// TwinCAT 3 PLC project mover_demo
// ProgramVersion: 3.1.4024.12
// libraries:
//   CmpBitmapPool, * (System)
//   Tc2_Math, * (Beckhoff Automation GmbH)
//   Tc2_MC2, * (Beckhoff Automation GmbH)
//   Tc2_MC2_Drive, * (Beckhoff Automation GmbH)
//   Tc2_Standard, * (Beckhoff Automation GmbH)
//   Tc2_System, * (Beckhoff Automation GmbH)
//   Tc2_Utilities, * (Beckhoff Automation GmbH)
//   Tc3_JsonXml, * (Beckhoff Automation GmbH)
//   Tc3_Module, * (Beckhoff Automation GmbH)
//   VisuDialogs, * (System)
//   VisuSymbols,3.5.10.0,System
// project tree:
//   DUTs/Helptec/Axis/ AxisBase_t.TcDUT (not stored), AxisBeckhoff_t.TcDUT (not stored), AxisLinMotConst_t.TcDUT, AxisLinMot_t.TcDUT (not stored), AxisSMC_t.TcDUT, typeInputArea.TcDUT, typeOutputArea.TcDUT (not stored)
//   DUTs/Helptec/ Cylinder2Pos_config.TcDUT (not stored), enLamp.TcDUT (not stored), enState.TcDUT (not stored), structAlarm.TcDUT (not stored), structButton.TcDUT (not stored)
//   DUTs/Helptec/Recipe/ RecipeAxisLinear2Pos_t.TcDUT (not stored)
//   DUTs/Helptec/RS_Axis/ FeederDelays_t.TcDUT, MoveProfile1D_t.TcDUT, MoveProfile_t.TcDUT (not stored), TriggerType_e.TcDUT (not stored), VectorMove1D_t.TcDUT (not stored)
//   DUTs/ PieceType_e.TcTLEO (not stored), Mover_st.TcDUT (not stored), Piece_st.TcDUT (not stored)
//   / GlobalTextList.TcGTLO (not stored) (excluded from build), PlcTask.TcTTO, Visualization Manager.TcVMO (not stored), VISU_TASK.TcTTO (not stored)
//   GVLs/ AXIS.TcGVL, CONST.TcGVL (not stored), GVL.TcGVL (not stored), HMI.TcGVL, IN.TcGVL (not stored), IO_BOX.TcGVL, OUT.TcGVL (not stored), PERS.TcGVL (not stored), SIMU.TcGVL (not stored)
//   POUs/00_MAIN/ DEBUG.TcPOU, MAIN.TcPOU, _02_SAFETY.TcPOU, _05_FLAGS.TcPOU (not stored)
//   POUs/00_MAIN/FB%27s/ FB_Safety.TcPOU (not stored)
//   POUs/10_HMI/FB%27s/ FB_BUTTON.TcPOU (not stored), FB_HMI_BT.TcPOU (not stored), FB_Keba_key.TcPOU (not stored), FB_LampeBNI007F.TcPOU (not stored), FB_STATE.TcPOU (not stored)
//   POUs/10_HMI/ _10_HMI.TcPOU (not stored), _11_PAR_CHK.TcPOU (not stored), _14_STATE.TcPOU (not stored)
//   POUs/20_AUTO/ Axis_e.TcTLEO, LinearAxis_e.TcTLEO (not stored), RecipeType_e.TcTLEO, Recipe_21_101_t.TcDUT (not stored), StationList_e.TcTLEO (not stored), _20_AUTO.TcPOU (not stored), _21_CopyDefaultRecipe.TcPOU (not stored)
//   POUs/20_AUTO/BuR SuperTrack com/ CT_Shuttle_BR_to_Tc_Status_t.TcDUT (not stored), CT_Shuttle_BR_to_Tc_t.TcDUT (not stored), CT_Shuttle_BR_to_Tc_u.TcDUT (not stored), CT_Shuttle_Tc_To_BR_Command_t.TcDUT (not stored), CT_Shuttle_Tc_to_BR_t.TcDUT, CT_Shuttle_Tc_to_BR_u.TcDUT, CT_Track_BR_to_TC_Status_t.TcDUT (not stored), CT_Track_BR_to_Tc_t.TcDUT (not stored), CT_Track_BR_to_Tc_u.TcDUT (not stored), CT_Track_Tc_to_BR_Command_t.TcDUT (not stored), CT_Track_Tc_to_BR_t.TcDUT, CT_Track_Tc_to_BR_u.TcDUT, gMoverAxis.TcGVL
//   POUs/20_AUTO/FB%27s/Alarm/ FB_ALARM.TcPOU (not stored), FB_ALARM32.TcPOU (not stored)
//   POUs/20_AUTO/FB%27s/ FB_WandlerForceSensor.TcPOU (not stored), getPercent.TcPOU (not stored)
//   POUs/20_AUTO/FB%27s/RS Axis/ BowlBandFeeder_Config_t.TcDUT (not stored), FB_AUT_Statistics.TcPOU (not stored), FB_BowlBandFeeder.TcPOU (not stored), FB_Feeder2Sensors.TcPOU (not stored), FB_Fifo.TcPOU (not stored), FB_LinearMotionMan.TcPOU (not stored), LinearMotionMan_Config_t.TcDUT (not stored)
//   POUs/20_AUTO/FB%27s/Achsen/ FB_AxisLIN_V1_1.TcPOU (not stored), FB_AxisLMturn_V1_1.TcPOU (not stored), FB_AxisLM_V1_1.TcPOU (not stored), FB_AxisRotTable_V1_1.TcPOU (not stored), FB_AxisSMC_V1_1.TcPOU (not stored), FB_AxisTURN_V1_1.TcPOU (not stored), JXCE1_Baustein.TcPOU (not stored)
//   POUs/20_AUTO/FB%27s/Pneumatic/ FB_ZylMo2El_V2_1.TcPOU (not stored)
//   POUs/20_AUTO/FB%27s/Vorlagen/ FB_ABL_VORLAGE.TcPOU (not stored), POU_AUT_VORLAGE.TcPOU (not stored), POU_ERR_VORLAGE.TcPOU (not stored), _01_MAIN.TcPOU (not stored)
//   POUs/20_AUTO/FileMan/ FB_FileMan.TcPOU (not stored), FileMan.TcPOU (not stored), LoadFromMemory.TcPOU, ReadJsonDom.TcPOU, SaveInMemory.TcPOU (not stored), SaveInMemory_Recipe.TcPOU (not stored)
//   POUs/20_AUTO/Mover/ ApproachScenario_e.TcTLEO (not stored), DistToTravel.TcPOU, FB_Group.TcPOU, FB_Mover.TcPOU (not stored), FB_MoverMan.TcPOU (not stored), FB_Position.TcPOU (not stored), FB_SimuMoverAxis.TcPOU (not stored), FB_Station.TcPOU (not stored), FB_PieceHolder.TcPOU (not stored), FB_StationMan.TcPOU, IProcessSampleMover.TcIO, ISimuMoverTimers.TcIO (not stored), IStation.TcIO (not stored), MoverDirection_e.TcTLEO (not stored), MoverState_e.TcTLEO, VISU_MoverDetail.TcVIS, VISU_MoverView.TcVIS (not stored), Pos2D_t.TcDUT (not stored), ProcessExec_e.TcDUT (not stored), StationName_e.TcTLEO
//   POUs/20_AUTO/Simu/ FB_Simu_AxisLIN_V1_1.TcPOU (not stored), FB_Simu_AxisLM_V1_1.TcPOU (not stored), FB_Simu_Feeder.TcPOU, FB_Simu_Zyl2Pos.TcPOU (not stored)
//   POUs/20_AUTO/ST100/ FB_ABL_LASER.TcPOU (not stored), FB_AUT_LASER.TcPOU (not stored), FB_AUT_100.TcPOU (not stored), F_GetPercent.TcPOU (not stored), F_GetPercent_2.TcPOU (not stored), ST100_Load_e.TcTLEO (not stored), FB_ABL_LOAD.TcPOU (not stored), FB_ABL_MODIFY.TcPOU (not stored), FB_ABL_UNLOAD.TcPOU (not stored), FB_AUT_ABSTRACT.TcPOU (not stored), FB_ABL_100.TcPOU (not stored), FB_AUT_LOAD.TcPOU, FB_AUT_MODIFY.TcPOU (not stored), FB_AUT_UNLOAD.TcPOU (not stored), ProcessExecution_e.TcTLEO (not stored), ST100_e.TcTLEO, ST100_Modify_e.TcTLEO (not stored), ST100_Laser_e.TcTLEO (not stored), ST100_Unload_e.TcTLEO (not stored)
//   POUs/20_AUTO/ST105/Fanuc_robot/ Fanuc_command_ext_to_robot_t.TcDUT (not stored), Fanuc_command_std_to_robot_t.TcDUT (not stored), Fanuc_hw_command_to_robot_t.TcDUT (not stored), Fanuc_status_std_from_robot.TcDUT, ST105_Fanuc_command_t.TcDUT (not stored), ST105_Fanuc_status_t.TcDUT (not stored)
//   POUs/20_AUTO/ST105/ FB_ABL_105_Feeder.TcPOU (not stored), FB_ABL_105_Pnp.TcPOU, FB_AUT_105.TcPOU (not stored), ST105_Axis.TcGVL (not stored), ST105_PnpVerPushPos_e.TcDUT (not stored), ST105_Recipe_t.TcDUT, ST105_Feeder_e.TcDUT (not stored), ST105_Pnp_e.TcTLEO (not stored), ST105_Slider_e.TcDUT (not stored), ST105_Cylinders_e.TcTLEO (not stored), VISU_Recipe_ST105.TcVIS (not stored), VISU_ST105.TcVIS (not stored)
//   POUs/20_AUTO/ST110/ POU_ALARM_110.TcPOU (not stored), ST110_Alarm_e.TcDUT, ST110_Cylinders_e.TcTLEO, ST110_Feeder_e.TcDUT (not stored), FB_ABL_110_Feeder.TcPOU (not stored), FB_ABL_110_Pnp.TcPOU (not stored), FB_AUT_110.TcPOU (not stored), ST110_Axis.TcGVL, ST110_PnpVerPushPos_e.TcDUT (not stored), ST110_Pnp_e.TcTLEO (not stored), ST110_PnpHorPos_e.TcDUT, ST110_PnpVerPos_e.TcDUT, ST110_Recipe_t.TcDUT, VISU_Recipe_ST110.TcVIS (not stored), VISU_ST110.TcVIS (not stored)
//   POUs/20_AUTO/ST115/ FB_ABL_115_Feeder.TcPOU (not stored), FB_ABL_115_Pnp.TcPOU (not stored), FB_AUT_115.TcPOU (not stored), ST115_PnpVerPushPos_e.TcDUT (not stored), ST115_Cylinders_e.TcTLEO (not stored), ST115_Recipe_t.TcDUT (not stored), ST115_Axis.TcGVL, ST115_Feeder_e.TcDUT (not stored), ST115_PnpHorPos_e.TcDUT (not stored), ST115_PnpVerPos_e.TcDUT, ST115_Pnp_e.TcTLEO (not stored), VISU_Recipe_ST115.TcVIS, VISU_ST115.TcVIS
//   POUs/20_AUTO/ST120/ FB_ABL_120_Feeder.TcPOU, FB_ABL_120_Pnp.TcPOU, FB_AUT_120.TcPOU (not stored), POU_ALARM_120.TcPOU, ST120_Alarm_e.TcDUT, ST120_Cylinders_e.TcTLEO (not stored), ST120_Axis.TcGVL (not stored), ST120_Feeder_e.TcDUT (not stored), ST120_PnpHorPos_e.TcDUT, ST120_PnpVerPos_e.TcDUT (not stored), ST120_Pnp_e.TcTLEO, ST120_Recipe_t.TcDUT (not stored), VISU_Recipe_ST120.TcVIS (not stored), VISU_ST120.TcVIS
//   POUs/20_AUTO/ST125/ FB_ABL_125_Feeder.TcPOU (not stored), FB_ABL_125_Pnp.TcPOU (not stored), FB_AUT_125.TcPOU (not stored), POU_ALARM_125.TcPOU (not stored), ST125_Alarm_e.TcDUT (not stored), ST125_Cylinders_e.TcTLEO (not stored), ST125_Axis.TcGVL (not stored), ST125_Feeder_e.TcDUT (not stored), ST125_PnpHorPos_e.TcDUT (not stored), ST125_PnpVerPos_e.TcDUT (not stored), ST125_Pnp_e.TcTLEO (not stored), ST125_Recipe_t.TcDUT (not stored), VISU_Recipe_ST125.TcVIS (not stored), VISU_ST125.TcVIS
//   POUs/20_AUTO/ST128/ FB_ABL_128_TubeCapCheck.TcPOU (not stored), FB_AUT_128.TcPOU, ST128_TubeCapCheck_e.TcTLEO, ST128_Recipe_t.TcDUT (not stored), VISU_Recipe_ST128.TcVIS, VISU_ST128.TcVIS (not stored)
//   POUs/20_AUTO/ST130/ FB_ABL_130_Dose.TcPOU (not stored), FB_ABL_MODIFY_135.TcPOU (not stored), FB_AUT_130.TcPOU (not stored), FB_AUT_135.TcPOU (not stored), ST130_Axis.TcGVL, ST130_Cylinders_e.TcTLEO, ST130_DosierkammerPos_e.TcDUT, ST130_PatroneAushebenPos_e.TcDUT (not stored), ST130_Recipe_t.TcDUT (not stored), ST130_Dose_e.TcTLEO (not stored), VISU_Recipe_ST130.TcVIS (not stored), VISU_ST130.TcVIS (not stored)
//   POUs/20_AUTO/ST140/ FB_ABL_140_Measure.TcPOU (not stored), FB_AUT_140.TcPOU, LaserPlace_e.TcDUT (not stored), ST140_Measure_e.TcTLEO (not stored), ST140_Recipe_t.TcDUT (not stored), VISU_Recipe_ST140.TcVIS, VISU_ST140.TcVIS (not stored)
//   POUs/20_AUTO/ST145/ FB_ABL_145_Feeder.TcPOU (not stored), FB_ABL_145_Pnp.TcPOU (not stored), FB_AUT_145.TcPOU, ST145_Axis.TcGVL, ST145_Cylinders_e.TcTLEO, ST145_Feeder_e.TcDUT (not stored), ST145_PnpHorPos_e.TcDUT, ST145_PnpVerPos_e.TcDUT (not stored), ST145_Recipe_t.TcDUT (not stored), ST145_Pnp_e.TcTLEO (not stored), VISU_Recipe_ST145.TcVIS (not stored), VISU_ST145.TcVIS (not stored)
//   POUs/20_AUTO/ST15x/ FB_ABL_150.TcPOU, FB_ABL_150_solo.TcPOU, FB_AUT_150.TcPOU (not stored), FB_AUT_155.TcPOU (not stored), ST150_Cylinders_e.TcTLEO (not stored), ST150_Uss_e.TcTLEO, ST150_Recipe_t.TcDUT, Ultrasonic_IN_bits_t.TcDUT (not stored), Ultrasonic_OUT_bits_t.TcDUT (not stored), VISU_Recipe_ST150.TcVIS (not stored), VISU_ST150.TcVIS (not stored)
//   POUs/20_AUTO/ST16x/CETA/ CETA_error_handling_t.TcDUT (not stored), CETA_IN_bits_t.TcDUT (not stored), CETA_IN_u.TcDUT (not stored), CETA_IO.TcGVL (not stored), CETA_OUT_bits_t.TcDUT (not stored), CETA_OUT_u.TcDUT (not stored), CETA_Result_e.TcDUT (not stored), CETA_Unit_e.TcDUT (not stored), FB_CETA_715.TcPOU (not stored)
//   POUs/20_AUTO/ST16x/CETA/CETA_Measurement_t/ CETA_Measurement_block1_t.TcDUT, CETA_Measurement_block2_t.TcDUT (not stored), CETA_Measurement_block3_t.TcDUT, CETA_Measurement_t.TcDUT (not stored), CETA_Res_Data_t.TcDUT (not stored)
//   POUs/20_AUTO/ST16x/CETA/CETA_Parameter_blocks/ CETA_Parameter_blocks_t.TcDUT (not stored)
//   POUs/20_AUTO/ST16x/CETA/CETA_com_union/ CETA_Parameter_blocks_u.TcDUT (not stored)
//   POUs/20_AUTO/ST16x/ FB_ABL_160.TcPOU, FB_AUT_160.TcPOU (not stored), FB_AUT_165.TcPOU (not stored), ST160_PnpVerPos_e.TcDUT (not stored), ST16x_Axis.TcGVL (not stored), ST160_Cylinders_e.TcTLEO (not stored), ST160_Recipe_t.TcDUT, ST160_CETA_e.TcTLEO (not stored), VISU_Recipe_ST160.TcVIS, VISU_ST160.TcVIS (not stored)
//   POUs/20_AUTO/ST170/ FB_ABL_170.TcPOU (not stored), FB_AUT_170.TcPOU (not stored), ST170_Axis.TcGVL, ST170_RFID_e.TcTLEO (not stored), ST170_PnpVerPos_e.TcDUT (not stored), ST170_Recipe_t.TcDUT (not stored), VISU_Recipe_ST170.TcVIS (not stored), VISU_ST170.TcVIS (not stored)
//   POUs/20_AUTO/ST175/ FB_ABL_175.TcPOU (not stored), FB_AUT_175.TcPOU (not stored), ST175_LASER_e.TcTLEO (not stored), ST175_Cylinders_e.TcTLEO (not stored), ST175_Recipe_t.TcDUT (not stored), VISU_Recipe_ST175.TcVIS, VISU_ST175.TcVIS
//   POUs/20_AUTO/ST175/Trumpf/ FB_Laser_ABL.TcPOU, if_BitCommand_u.TcDUT, if_Command_t.TcDUT (not stored), if_Command_u.TcDUT (not stored), if_SingleCmds.TcGVL (not stored), if_TruMark.TcGVL (not stored), TruMarkLaserStatus.TcDUT (not stored), TruMark_Ethercat_dj.TcPOU (not stored), TruMark_SingleCmds.TcPOU (not stored)
//   POUs/20_AUTO/ST180/ FB_ABL_180_Pnp.TcPOU (not stored), FB_AUT_180.TcPOU (not stored), ST180_Axis.TcGVL (not stored), ST180_Cylinders_e.TcTLEO (not stored), ST180_PnpHorPos_e.TcDUT, ST180_PnpVerPos_e.TcDUT, ST180_Pnp_e.TcTLEO (not stored), ST180_Recipe_t.TcDUT (not stored), VISU_Recipe_ST180.TcVIS (not stored), VISU_ST180.TcVIS
//   POUs/20_AUTO/ST185/ FB_ABL_185_Pnp.TcPOU (not stored), FB_AUT_185.TcPOU (not stored), ST185_Axis.TcGVL (not stored), ST185_Cylinders_e.TcTLEO (not stored), ST185_PnpHorPos_e.TcDUT (not stored), ST185_PnpVerPos_e.TcDUT (not stored), ST185_Pnp_e.TcTLEO (not stored), ST185_Recipe_t.TcDUT (not stored), VISU_Recipe_ST185.TcVIS (not stored), VISU_ST185.TcVIS
//   POUs/20_AUTO/TOOL/ ASSERT.TcPOU (not stored), EqualApproximately.TcPOU (not stored), EqualDelta.TcPOU (not stored), EqualEssentially.TcPOU (not stored), GetTick.TcPOU (not stored), IObject.TcIO (not stored), MAP_REAL_TO_INT.TcPOU (not stored), SortBubbleLREAL.TcPOU (not stored)
//   VISUs/ Custom.TcIPO (not stored), VISU_LinearConfigArray.TcVIS (not stored), VISU_Cylinder2PosConfig.TcVIS (not stored), VISU_AxisManual.TcVIS (not stored), VISU_main.TcVIS (not stored), VISU_Time.TcVIS (not stored)

CONFIGURATION mover_demo
    RESOURCE PLC ON TwinCAT3
        TASK PlcTask(INTERVAL := T#10ms, PRIORITY := 20);
        PROGRAM MAIN WITH PlcTask : MAIN;
        PROGRAM TruMark_Ethercat_dj WITH PlcTask : TruMark_Ethercat_dj;
        PROGRAM TruMark_SingleCmds WITH PlcTask : TruMark_SingleCmds;
    END_RESOURCE
END_CONFIGURATION

// ---- DUTs/Helptec/Axis/AxisLinMotConst_t.TcDUT
TYPE AxisLinMotConst_t :
STRUCT
    POS_MIN   : REAL; // Software limit switch of the minimum position
    POS_MAX   : REAL; // Software limit switch of the maximum position
    VELO_MAX  : REAL; // Maximum allowed velocity
    VELO_MANU : REAL; // Velocity in manual mode
END_STRUCT
END_TYPE

// ---- DUTs/Helptec/Axis/AxisSMC_t.TcDUT
TYPE AxisSMC_t EXTENDS AxisBase_t :
STRUCT
    typeOUT AT %Q* : typeOutputArea; // Axis reference SMC output
    typeIN  AT %I* : typeInputArea;  // Axis reference SMC input
END_STRUCT
END_TYPE

// ---- DUTs/Helptec/Axis/typeInputArea.TcDUT
TYPE typeInputArea :
STRUCT
    SigAllToTheInpPor         : UINT;
    ControllerInformationFlag : UINT;
    CurrentPosition           : DINT;
    CurrentSpeed              : UINT;
    CurrentPushForce          : UINT;
    TargetPosition            : DINT;
    Alarm1                    : USINT;
    Alarm2                    : USINT;
    Alarm3                    : USINT;
    Alarm4                    : USINT;
END_STRUCT
END_TYPE

// ---- DUTs/Helptec/RS_Axis/FeederDelays_t.TcDUT
TYPE FeederDelays_t :
STRUCT
    InFilterDelay : DINT; // delay to filter the input, see FB_Feeder2Sensors
    StartDelay    : DINT; // delay to start the feeder, see FB_Feeder2Sensors
    StopDelay     : DINT; // delay to stop the feeder, see FB_Feeder2Sensors
    EmptyDelay    : DINT; // delay before the feeder is considered as empty, see FB_Feeder2Sensors
END_STRUCT
END_TYPE

// ---- DUTs/Helptec/RS_Axis/MoveProfile1D_t.TcDUT
// Specify a 1D mouvement, the position only represents a point in the 1D space
TYPE MoveProfile1D_t :
STRUCT
    lrVelocity : REAL;  // Velocity to position
    lrAccel    : REAL;  // acceleration to position
    lrDecel    : REAL;  // deceleration to position
    lrJerk     : REAL;  // jerk to position
    lrPosition : LREAL; // Position to go
END_STRUCT
END_TYPE

// ---- POUs/20_AUTO/Axis_e.TcTLEO
{attribute 'qualified_only'}
{attribute 'strict'}
{attribute 'to_string'}
TYPE Axis_e :
(
	ST105_10W,  //  0
	ST105_11Z,  //  1
    ST110_01Y,  //  2
    ST110_02Z,  //  3
    ST110_03Z,  //  4
    ST110_04Z,  //  5
	ST110_10W,  //  6
    ST115_01Y,  //  7
    ST115_02Z,  //  8
    ST115_03Z,  //  9
    ST115_04Z,  // 10
	ST115_10W,  // 11
    ST120_01Y,  // 12
    ST120_02Z,  // 13
    ST125_01Y,  // 14
    ST125_02Z,  // 15
	ST125_10W,  // 16
	ST130_01Z,  // 17
	ST130_10Z,  // 18
	ST135_01Z,  // 19
	ST135_10Z,  // 20
	ST145_01Y,  // 21
	ST145_02Z,  // 22
	ST145_10W,  // 23
	ST160_01Z,  // 24
	ST165_01Z,  // 25
	ST170_01Z,  // 26
	ST180_01Y,  // 27
	ST180_02Z,  // 28
	ST180_10Z,  // 29
	ST185_01Y,  // 30
	ST185_02Z,  // 31
	ST185_10Z,  // 32
    _max
);
END_TYPE

// ---- POUs/20_AUTO/BuR SuperTrack com/CT_Shuttle_Tc_to_BR_t.TcDUT
{attribute 'pack_mode' := '1'}
TYPE CT_Shuttle_Tc_to_BR_t :
STRUCT
    bCommand        : CT_Shuttle_Tc_To_BR_Command_t; (* command bit field *)
    bNextStation    : BYTE; (* next station *)
    diNextOffset_um : DINT; (* 4 byte value that represent the offset in um. This value needs to be between -500'000 and 500'000 um *)
END_STRUCT
END_TYPE

// ---- POUs/20_AUTO/BuR SuperTrack com/CT_Shuttle_Tc_to_BR_u.TcDUT
{attribute 'pack_mode' := '1'}
TYPE CT_Shuttle_Tc_to_BR_u :
UNION
    asStruct : ARRAY[1..20] OF CT_Shuttle_Tc_to_BR_t;
    asArray  : ARRAY[0..20 * SIZEOF(CT_Shuttle_Tc_to_BR_t) - 1] OF USINT;
END_UNION
END_TYPE

// ---- POUs/20_AUTO/BuR SuperTrack com/CT_Track_Tc_to_BR_t.TcDUT
{attribute 'pack_mode' := '1'}
TYPE CT_Track_Tc_to_BR_t :
STRUCT
    bCommand : CT_Track_TC_to_BR_Command_t; (* command bit field for the track system *)
END_STRUCT
END_TYPE

// ---- POUs/20_AUTO/BuR SuperTrack com/CT_Track_Tc_to_BR_u.TcDUT
{attribute 'pack_mode' := '1'}
TYPE CT_Track_Tc_to_BR_u :
UNION
    asStruct : CT_Track_Tc_to_BR_t;
    asArray  : ARRAY[0..SIZEOF(CT_Track_Tc_to_BR_t)-1] OF USINT;
END_UNION
END_TYPE

// ---- POUs/20_AUTO/RecipeType_e.TcTLEO
{attribute 'qualified_only'}
{attribute 'strict'}
TYPE RecipeType_e :
(
    Smart := 0,
    Pro := 1,
    Mini := 2,
    Blue := 3,
    Smart_Kristall := 4,
    Pro_Smart := 5,
    Pro_Blue := 6,
    Pro_Smart_Kristall := 7,
    Pro_Smart_Maxi := 8,
    Pro_Smart_Maxi_Kristall := 9,
    Reserve := 10,
    _max
);
END_TYPE

// ---- POUs/20_AUTO/Mover/MoverState_e.TcTLEO
{attribute 'qualified_only'}
{attribute 'strict'}
{attribute 'to_string'}
TYPE
MoverState_e :
(
    OperationDone,           // The operation on the mover is done, a new station needs to be given
    WaitOnNextStation,       // wait on the next station to be ready. The waiting depend on the scenario of the next station
    WaitLeaveCurrentStation, // If we are bind with the track system, we will be sure that we have actualy leaved the curent station
    MovingToStation,         // the mover is moving or try to move to the next station
    InStationPos,            // The mover is currently AT the station position (aka target pos.), waiting on the process TO begin
    InOperation,             // The attached process of the mover is running. The mover is not able to move
    PerformRelativeMove,     // Moving the mover when already in operation, go to WaitRelativeMoveEnd when mover actually moving
    WaitRelativeMoveEnd,     // Wait on the At_pos flag
    _MAX
);
END_TYPE

// ---- POUs/20_AUTO/Mover/StationName_e.TcTLEO
{attribute 'qualified_only'}
{attribute 'to_string'}
TYPE
StationName_e :
(
    Station_105 := 1,
    Station_110 := 2,
    Station_115 := 3,
    Station_120 := 4,
    Station_125 := 5,
    Station_130 := 6,
    Station_135 := 7,
    Station_140 := 8,
    Station_145 := 9,
    Station_150 := 10,
    Station_155 := 11,
    Station_160 := 12,
    Station_165 := 13,
    Station_170 := 14,
    Station_175 := 15,
    Station_176 := 16,
    Station_180 := 17,
    Station_185 := 18
);
END_TYPE

// ---- POUs/20_AUTO/ST100/ST100_e.TcTLEO
{attribute 'qualified_only'}
{attribute 'strict'}
{attribute 'to_string'}
TYPE
ST100_e :
(
    RESET := 0,         // Reset
    INIT := 100,        // Initialisieren
	
	
	
    READY := 999,       // READY to Start, Init Done 
    START := 1000,      // Start Zyklisch
    MOVER_FREE_OP,      // Ab here, operation without mover can be done
    proceedOperation_1, //proceed to some operation
    waitOnMover,        // wait until the mover is there
    MOVER_NEEDED_OP,    // Ab here, a mover in position is needed to perform the action
    proceedOperation_2, //proceed to some operation
    DONE := 8000,       // Ablauf beendet 
    ERROR := 9000,      // Fehler 
    _max
);
END_TYPE


// 0:  // setup everything
// 5:  // wait until the whole path is free
// 10: // turn power on
// 11: // init all mover until they the first shuttle is found
// 12: // set all id since the first is found
// 13: // stop id attrib sequence                
// 14: // check parameter
// 15: //move every shuttle to the last station
// 16: // do nothing, init done

// ---- POUs/20_AUTO/ST105/Fanuc_robot/Fanuc_status_std_from_robot.TcDUT
TYPE Fanuc_status_std_from_robot :
STRUCT
    CMD_enable   : BIT;
    SYSTEM_Ready : BIT;
    PRG_Running  : BIT;
    Prg_Paused   : BIT;
    Motion_Held  : BIT;
    Fault        : BIT;
    AT_Perch     : BIT;
    TP_enabled   : BIT;
    Batt_Alarm   : BIT;
    Busy         : BIT;
    Ack1_SNO1    : BIT;
    Ack2_SNO2    : BIT;
    Ack3_SNO3    : BIT;
    Ack4_SNO4    : BIT;
    Ack5_SNO5    : BIT;
    Ack6_SNO6    : BIT;
    Ack7_SNO7    : BIT;
    Ack8_SNO8    : BIT;
    SNACK        : BIT;
    RESERVED     : BIT;
END_STRUCT
END_TYPE

// ---- POUs/20_AUTO/ST105/ST105_Recipe_t.TcDUT
TYPE ST105_Recipe_t :
STRUCT
    xUseVerLeft        : BOOL; // Is the left vertical picker element is used
    xUseVerRight       : BOOL; // Is the right vertical picker element is used
    FeederConfig       : FeederDelays_t;
    FeederSize         : DINT; // tell the feeder slots number, if it has 2 slots or 
    PickOffset_X_deci  : UINT; // X offset of picking position
    PickOffset_Y_deci  : UINT; // Y offset of picking position
    PickUpPos_Z_deci   : UINT; // Z traveling height from pick to place position
    isPickOffset_X_neg : BOOL; // tell the robot that PickOffset_X_deci is negative
    isPickOffset_Y_neg : BOOL; // tell the robot that PickOffset_Y_deci is negative
    isPickUpPos_Z_neg  : BOOL; // tell the robot that PickUpPos_Z_deci is negative
END_STRUCT
END_TYPE

// ---- POUs/20_AUTO/ST110/ST110_Alarm_e.TcDUT
{attribute 'qualified_only'}
{attribute 'to_string'}
TYPE ST110_Alarm_e :
(
    no_error := 0,
    Axis_110_01Y_error := 1,
    Axis_110_02Z_error := 2,
    Axis_110_03Z_error := 3,
    Axis_110_04Z_error := 4,
    Cylinder_vacuum_griper_left := 5,
    Cylinder_vacuum_griper_right := 6,
    Axis_110_10W_error := 7,
    Feeder_error := 8,
    Piece_in_unused_griper := 9,
    Piece_missing_left_griper := 10,
    Piece_missing_right_griper := 11,
    Feeder_empty := 12,
	Reach_end_pos_without_needed_torque := 13,
    _max := 20
)BYTE;
END_TYPE

// ---- POUs/20_AUTO/ST110/ST110_Cylinders_e.TcTLEO
{attribute 'qualified_only'}
{attribute 'strict'}
{attribute 'to_string'}
TYPE ST110_Cylinders_e :
(
    VakuumgreiferLinks,
    VakuumgreiferRechts,
    _max
);
END_TYPE

// ---- POUs/20_AUTO/ST110/ST110_PnpHorPos_e.TcDUT
{attribute 'qualified_only'}
{attribute 'to_string'}
TYPE ST110_PnpHorPos_e :
(
	GS,
	AS,
	_max
);
END_TYPE

// ---- POUs/20_AUTO/ST110/ST110_PnpVerPos_e.TcDUT
{attribute 'qualified_only'}
{attribute 'to_string'}
TYPE ST110_PnpVerPos_e :
(
    UpEmpty,               // Up position when the Pnp is empty
    DownEmpty,             // Down position when the Pnp is picking the piece
    UpFull,                // Up position when the Pnp has gripped the piece
    DownFullQuick,         // down position with quick speed
    DownFullTorqueControl, // down position with low speed for torque control
    _max
);
END_TYPE

// ---- POUs/20_AUTO/ST110/ST110_Recipe_t.TcDUT
TYPE ST110_Recipe_t :
STRUCT
    xUseVerLeft         : BOOL; // Is the left vertical picker element is used
    xUseVerRight        : BOOL; // Is the right vertical picker element is used
    FeederConfig        : FeederDelays_t;
    waitBlowPieceTon_ms : DINT; // time to wait before to blow the piece away
    blowPieceTof_ms     : DINT; // time to let the blower take away the piece
    vakum_left_pc       : INT;  // vacum limit for left pnp
    vakum_right_pc      : INT;  // vacum limit for right pnp
    kraft_left_raw      : REAL;  // force limit for left pnp, raw value
    kraft_right_raw     : REAL;  // force limit for right pnp, raw value
END_STRUCT
END_TYPE

// ---- POUs/20_AUTO/ST115/ST115_PnpVerPos_e.TcDUT

TYPE ST115_PnpVerPos_e : ST110_PnpVerPos_e;
END_TYPE

// ---- POUs/20_AUTO/ST120/ST120_Alarm_e.TcDUT
{attribute 'qualified_only'}
{attribute 'to_string'}
TYPE ST120_Alarm_e :
(
    no_error := 0,
    Axis_120_01Y_error := 1,
    Axis_120_02Z_error := 2,
    Cylinder_griper_left := 3,
    Cylinder_griper_right := 4,
    Cylinder_pivot_left := 5,
    Cylinder_pivot_right := 6,
    Cylinder_hublader_left := 7,
    Cylinder_hublader_right := 8,
    Piece_in_unused_griper := 9,
    Piece_missing_left_griper := 10,
    Piece_missing_right_griper := 11,
    Feeder_empty := 12,
    Feeder_error := 13,
    Piece_in_unused_pivot := 14,
    Piece_missing_left_pivot := 15,
    Piece_missing_right_pivor := 16,
	
    _max := 20
) BYTE;
END_TYPE

// ---- POUs/20_AUTO/ST120/ST120_PnpHorPos_e.TcDUT
TYPE ST120_PnpHorPos_e : ST110_PnpHorPos_e;
END_TYPE

// ---- POUs/20_AUTO/ST120/ST120_Pnp_e.TcTLEO
{attribute 'qualified_only'}
{attribute 'strict'}
{attribute 'to_string'}
TYPE ST120_Pnp_e :
(
    RESET := 0, // Reset

    INIT := 100, // Initialisieren 
    Init_HomeVerticals,
    Init_VerticalsUp,
    Init_HomeHorizontals,
    Init_HorizontalsToTrack,
    Init_adjust_left_clamp,
    Init_open_left_clamp,
    Init_adjust_right_clamp,
    Init_open_right_clamp,
    Init_check_if_pces_handled,

    MOVER_FREE_OP, // Ab here, operation without mover can be done
    READY := 999,  // READY to Start, Init Done 
    START := 1000, // Start Zyklisch

    PnP_Hor_ToRotTablePos,
    PnP_WaitOnFeeder,
    PnP_Ver_RotTableDown,
    Gripper_close,
    PnP_Ver_RotTableUp,
    PnP_Hor_ToTrackPos,
    waitOnMover,     // wait until the mover is there
    MOVER_NEEDED_OP, // Since here, a mover in position is needed to perform the action

    PnP_Ver_ShuttleDown,
    PnP_Ver_ShuttleTorqueControl,
    Gripper_open,
    PnP_Ver_ShuttleUp,

    SYNC_MOVER_LEAVE, // MoverMan need to take the mover
    DONE := 8000,     // Ablauf beendet 
    ERROR := 9000,    // Fehler 
    _max
);
END_TYPE

// ---- POUs/20_AUTO/ST128/ST128_TubeCapCheck_e.TcTLEO
{attribute 'qualified_only'}
{attribute 'strict'}
{attribute 'to_string'}
TYPE
ST128_TubeCapCheck_e :
(
    RESET := 0, // Reset

    INIT := 100, // Initialisieren 

    READY := 999,  // READY to Start, Init Done 
    START := 1000, // Start Zyklisch

    waitOnMover,     // wait until the mover is there
    MOVER_NEEDED_OP, // Ab here, a mover in position is needed to perform the action

    Move_shuttle_relative_right,
	Wait_move_and_check_tube_cap_right,
    Move_shuttle_to_pos_left,
	Wait_move_done_pos_left,
    Move_shuttle_relative_left,
	Wait_move_and_check_tube_cap_left,
    Save_result_in_mover,

    SYNC_MOVER_LEAVE, // MoverMan need to take the mover
    MOVER_FREE_OP,    // here, operation without mover can be done.

    DONE := 8000,  // Ablauf beendet 
    ERROR := 9000, // Fehler 
    _max
);
END_TYPE

(*
back to shuttle
check level NIO Box
*)

// ---- POUs/20_AUTO/ST130/ST130_Cylinders_e.TcTLEO
{attribute 'qualified_only'}
{attribute 'strict'}
{attribute 'to_string'}
TYPE ST130_Cylinders_e :
(
    Kammer_Offnen_Links,
    Kammer_Offnen_Rechts,
    Kammer_nachfullen_Links,
    Kammer_nachfullen_Rechts,
    Vibrieren_Kammer_Links,
    Vibrieren_Kammer_Rechts,
    Niederhalter_Patrone,
    Vibrienren_Patrone_Links,
    Viebrieren_Patrone_Rechts
);
END_TYPE

// ---- POUs/20_AUTO/ST130/ST130_DosierkammerPos_e.TcDUT
TYPE ST130_DosierkammerPos_e :
(
    up_GS,
    down_AS,
    _max
);
END_TYPE

// ---- POUs/20_AUTO/ST145/ST145_Cylinders_e.TcTLEO
TYPE ST145_Cylinders_e : ST110_Cylinders_e;
END_TYPE

// ---- POUs/20_AUTO/ST145/ST145_PnpHorPos_e.TcDUT
{attribute 'qualified_only'}
{attribute 'strict'}
{attribute 'to_string'}
TYPE ST145_PnpHorPos_e :
(
    GS_After_placement,
    GS_Before_placement,
    AS_to_feeder,
    _max
);
END_TYPE

// ---- POUs/20_AUTO/ST15x/ST150_Uss_e.TcTLEO
{attribute 'qualified_only'}
{attribute 'strict'}
{attribute 'to_string'}
TYPE ST150_Uss_e :
(
    RESET := 0, // Reset

    INIT := 100, // Initialisieren 
    Init_ResetUss_maintaining_down,

    READY := 999,  // READY to Start, Init Done 
    START := 1000, // Start Zyklisch

    waitOnMover,     // wait until the mover is there
    MOVER_NEEDED_OP, // Since here, a mover in position is needed to perform the action

    check_cap_present,     // See if the sensor sees the cap
    mover_maintening_up,   // Kraftbstützung goes up
    uss_start,             // start signal is given
    uss_working,           // we wait until the uss is finished
    mover_maintening_down, // Kraftbstützung goes down

    // only used for xxxx_solo process
    move_shuttle_120_mm,
    wait_shuttle_in_pos,

    SYNC_MOVER_LEAVE, // MoverMan need to take the mover
    MOVER_FREE_OP,    // Ab here, operation without mover can be done

    DONE := 8000,  // Ablauf beendet 
    ERROR := 9000, // Fehler 
    _max
);
END_TYPE

// ---- POUs/20_AUTO/ST15x/ST150_Recipe_t.TcDUT
TYPE ST150_Recipe_t :
STRUCT
    USS_ErrorTime_ms : DINT; // timeout of the start signal
    USS_Type         : SINT; // byte code to send to the USS before welding
END_STRUCT
END_TYPE

// ---- POUs/20_AUTO/ST16x/CETA/CETA_Measurement_t/CETA_Measurement_block1_t.TcDUT
{attribute 'pack_mode' := '1'}
TYPE CETA_Measurement_block1_t :
STRUCT
    Program_number : USINT;
    Result         : USINT;
    Test_mode      : USINT;
    Date_day       : USINT;
    Date_month     : USINT;
    Date_year      : USINT;
    Date_century   : USINT;
    Time_hour      : USINT;
    Time_minute    : USINT;
    Time_second    : USINT;
    Data_offset_12 : CETA_Res_Data_t;
    Data_offset_16 : CETA_Res_Data_t;
    Data_offset_20 : CETA_Res_Data_t;
    Data_offset_24 : CETA_Res_Data_t;
    Data_offset_28 : CETA_Res_Data_t;
    Data_offset_32 : CETA_Res_Data_t;
    Data_offset_36 : CETA_Res_Data_t;
    Data_offset_40 : CETA_Res_Data_t;
    Data_offset_44 : CETA_Res_Data_t;
    Data_offset_48 : CETA_Res_Data_t;
    Data_offset_52 : CETA_Res_Data_t;
    Data_offset_56 : CETA_Res_Data_t;
    Data_offset_60 : CETA_Res_Data_t;
END_STRUCT
END_TYPE

// ---- POUs/20_AUTO/ST16x/CETA/CETA_Measurement_t/CETA_Measurement_block3_t.TcDUT
{attribute 'pack_mode' := '1'}
TYPE CETA_Measurement_block3_t :
STRUCT
    Program_number       : USINT;
    Result_chanel_1      : USINT;
    Test_mode            : USINT;
    Result_chanel_2      : USINT;
    Cons_Num_Res_Block   : USINT;
    Num_Following_Blocks : USINT;
    Reserve              : USINT;
    Time_hour            : USINT;
    Time_minute          : USINT;
    Time_second          : USINT;
    Data_offset_12       : CETA_Res_Data_t;
    Data_offset_16       : CETA_Res_Data_t;
    Data_offset_20       : CETA_Res_Data_t;
    Data_offset_24       : CETA_Res_Data_t;
END_STRUCT
END_TYPE

// ---- POUs/20_AUTO/ST16x/ST160_Recipe_t.TcDUT
TYPE ST160_Recipe_t :
STRUCT
    Use_element_left  : BOOL; //a 
    Use_element_right : BOOL; // 
    Program_number    : USINT; // 
END_STRUCT
END_TYPE

// ---- POUs/20_AUTO/ST175/Trumpf/if_BitCommand_u.TcDUT
TYPE if_BitCommand_u :
UNION
    awPBOM : ARRAY[0..1] OF WORD;
    dwPBOM : DWORD;
END_UNION
END_TYPE

// ---- POUs/20_AUTO/ST180/ST180_PnpHorPos_e.TcDUT
TYPE ST180_PnpHorPos_e : ST110_PnpHorPos_e;
END_TYPE

// ---- POUs/20_AUTO/ST180/ST180_PnpVerPos_e.TcDUT
TYPE ST180_PnpVerPos_e :
(
    up_waiting_mover,
    down_empty,
    up_full,
    down_full,
	up_after_unload,
    _max
);
END_TYPE

// ---- GVLs/AXIS.TcGVL
{attribute 'qualified_only'}
(*******************************************************************)
(* ACHSEN KONSTANTEN *)
(*******************************************************************)
VAR_GLOBAL CONSTANT

END_VAR
VAR_GLOBAL
    (*******************************************************************)
    (* ACHSEN Variablen *)
    (*******************************************************************)
    //Axis Allgemein Teachen und Anzeige
    bTeachAxisNr  : BYTE;                              // Zu Teachende Achse # (von HMI)
    bTeachInPos   : BYTE;                              // Achse in Position (Teachpos (99= nicht in Pos))
    bTeachPos     : ARRAY[0..Axis_e._max - 1] OF BYTE; // Achse Teach Position (Anzufahrende Position #)
    rTeachIncAxis : REAL := 0.1;                       // Axis Inching Wert
    rTeachVelo    : REAL := 10;                        // Achse Geschwindigkeit (Anzeige)
    rTeachPos     : REAL;                              // Achse Teach Position (Anzufahrende Position Wert)
    rTeachActPos  : REAL;                              // Achse AKTUELLE Position (AKTUEL
    rTeachPosMin  : REAL;                              // Achse PositionsminimumLER Position Wert)
    rTeachPosMax  : REAL;                              // Achse Positionsmaximum
    rJogVelo_pc   : REAL                := REAL#10.0;  // global jog velocity in pc
    arrJogValues  : ARRAY[0..7] OF REAL := [0.01,      // lookup table for jog % value
                                            0.05,
                                            0.1,
                                            0.5,
                                            1.0,
                                            5.0,
                                            10.0,
                                            50.0];

    btTeachArAxis : ARRAY[0..Axis_e._max - 1] OF ARRAY[0..8] OF structButton; (* Buttons AXIS
                                                    0: Disable 
                                                    1: Inching 
                                                    2: Slow 
                                                    3: Fast 
                                                    4: Move Abs/Rel   
                                                    5: Manu Move NEGATIVE
                                                    6: Manu Move POSITIVE  
													7: Start Homing 
													8: Teachpos Übernehmen*)
END_VAR

(*******************************************************************)
(* ACHSEN Positionen von HMI*)
(*******************************************************************)
VAR_GLOBAL RETAIN

END_VAR

// ---- GVLs/HMI.TcGVL
{attribute 'qualified_only'}
VAR_GLOBAL
    (*******************************************************************)
    (* Globale HMI Variablen *)
    (*******************************************************************)
    xImmer0 : BOOL := FALSE; //ALLWAYS FALSE
    xImmer1 : BOOL := TRUE;  //ALLWAYS TRUE

    (*******************************************************************)
    (* Flags *)
    (*******************************************************************)
    enState   : enState; //SYSTEM STATUS
    xInitDone : BOOL;    //SYSTEM INITIALIZED
    xRefDone  : BOOL;    //Axis REF
    xAlarm    : BOOL;    //ALARM AKTIV
    xMessage  : BOOL;    //MELDUNG AKTIV
    xWait     : BOOL;    //ALLE FBs warten
    xAIRon    : BOOL;    //Luftdruck IO
    xSPC      : BOOL;    //SPC angewählt

    Tast_BL : BOOL; // ... 

    (*******************************************************************)
    (* Buttons *)
    (*******************************************************************)
    //Control
    btArMain : ARRAY[0..20] OF structButton; (*	
													0: AUTO
													1: STEP
													2: END
													3: MANU
													4: INIT
													5: STOP
													6: LEER
													7: QUIT
													8: RESET TEMP COUNTER
													9: START
													10: HUBTÜREn ALLE
													11: HUBTÜRE 1
													12: HUBTÜRE 2
													13: HUBTÜRE 3
													14: HUBTÜRE 4
												*)
    //Manual pneumatics
    // see below for button button instance 
    btManuCylinders : ARRAY[0..StationList_e._max] OF ARRAY[0..CONST.MAX_CYLINDER_PER_STATION] OF structButton;
    (* 
	 * [StationList_e.ST105] 0
     * [0]: Zyklus [1]: Robot get [2]: Robot set [3] Feeder
	 *
     * [StationList_e.ST110] 1
     * [0]: Zyklus [1]: Vacum Gripper left [2]: Vacum Gripper right [3]: Feeder
     *
     * [StationList_e.ST115] 2
     * [0]: Zyklus [1]: Gripper left [2]: Gripper right [3]: Feeder
     *
     * [StationList_e.ST120] 3
     * [0]: Zyklus [1]: Gripper left [2]: Gripper right [3]: Rotative cylinder left
     * [4]: Rotative cylinder right [5]: Hublader left [6]: Hublader right
	 * [7]: feeder left [8]: feeder right
     *
     * [StationList_e.ST125] 4
     * [0]: Zyklus [1]: Gripper left [2]: Gripper right [3]: lock cylinder left
     * [4]: lock cylinder right [5]: Gripper Solerohr left [6]: Gripper Solerohr right
	 * [7]: feeder 
     *
     * [StationList_e.ST130] 5
     * [0]: Zyklus [1]: cell open left [2]: cell open right [3]: cell fill left
     * [4]: cell fill right [5]: vib cell left [6]: vib cell right
	 * [7]: holder patrone [8]: vib patrone left [9]: vib patrone right [10]: Feeder 
     *
     * [StationList_e.ST135] 6
	 * dito ST130
	 *
     * [StationList_e.ST145] 8
     * [0]: Zyklus [1]: Vacum Gripper left [2]: Vacum Gripper right [3]: Feeder
	 *
     * [StationList_e.ST150] 9
     * [0]: Zyklus [1]: mover maintening [2]: start welding
	 *
     * [StationList_e.ST155] 10
     * [0]: Zyklus [1]: mover maintening [2]: start welding
	 *
     * [StationList_e.ST160] 11
     * [0]: Zyklus [1]: holder left [2]: holder right [3]: seal left
	 * [4]: seal right [5]: fill left [6]: fill right [7]: start test
	 *
     * [StationList_e.ST165] 12
     * [0]: Zyklus [1]: holder left [2]: holder right [3]: seal left
	 * [4]: seal right [5]: fill left [6]: fill right [7]: start test
	 *
     * [StationList_e.ST170] 13
     * [0]: Zyklus [1]: start test left [2]: start test right
	 *
     * [StationList_e.ST175] 14
     * [0]: Zyklus [1]: holder [2]: cabine in [3]: cabine out
	 * [4]: start laser
	 *
     * [StationList_e.ST180] 15
     * [0]: Zyklus [1]: Gripper left [2]: Gripper right 
	 * [3]: holder left [4]: holder right
	 *
     * [StationList_e.ST185] 11
     * [0]: Zyklus [1]:  [2]: 
     *)

    btArST150 : ARRAY[0..20] OF structButton; (*	0 : Start USS
	                                                1 : Reset US
											   *)

    btArForceCyclus     : ARRAY[0..StationList_e._max - 1] OF structButton;
    bArForceCyclusState : ARRAY[0..StationList_e._max - 1] OF BOOL;

    (*******************************************************************)
    (* ALARME  *)
    (*******************************************************************)
    strArALARM  : ARRAY[1..500] OF structAlarm;
    strArMSG    : ARRAY[1..100] OF structAlarm;
    xArAlarmHMI : ARRAY[1..9999] OF BOOL;

    (*******************************************************************)
    (* ANZEIGE - Werte *)
    (*******************************************************************)
    iSelectAxis     : LinearAxis_e := LinearAxis_e.ST110_01Y;
    iSelectAxisCopy : LinearAxis_e := LinearAxis_e._max;
    btCopyAxisCfg   : structButton;

    iSelectCylinder     : StationList_e := StationList_e.ST105;
    iSelectCylinderCopy : StationList_e := StationList_e._max;
    btCopyCylinderCfg   : structButton;

    iSelectJogAxis : Axis_e;

    (*******************************************************************)
    (* Cycle Time [STATION]*)
    (*******************************************************************)
    dwArStartTime_ms : ARRAY[0..StationList_e._max - 1] OF DWORD;
    dwArCycleTime_ms : ARRAY[0..StationList_e._max - 1] OF DWORD;

    lrPiecePerMinute : LREAL;

    PieceDoneTmp : DINT; // number of piece done since last reset

    (*******************************************************************)
    (* Recipe HMI management *)
    (*******************************************************************)
    btCopyRecipe  : structButton;
    btSetDefault  : structButton;
    movesNames    : ARRAY[0..LinearAxis_e._max - 1] OF ARRAY[0..CONST.MAX_VECTOR_LIST] OF STRING;
    cylinderNames : ARRAY[0..StationList_e._max - 1] OF ARRAY[0..CONST.MAX_CYLINDER_PER_STATION] OF STRING;

    (*******************************************************************)
    (* Mover manual bt *)
    (*******************************************************************)
    selectedShuttle : INT := 1; // selected shuttle from the HMI

    (*******************************************************************)
    (* Diverses *)
    (*******************************************************************)
    xWriteALlog : BOOL;         // Alarmlog schreiben in File
    btWritePers : structButton; // write pers data in filesystem

    sCurrentHMI2 : STRING; // ???
END_VAR

// ---- GVLs/IO_BOX.TcGVL
{attribute 'qualified_only'}
VAR_GLOBAL
    (*******************************************************************)
    (* EINGÄNGE Schrank A *)
    (*******************************************************************)

    (* IO-Link Boxen 190A1 *)
    (*******************************************************************)
    //-194A3
    (* BN Lampe *)
    Q0000_Balluf_Lampe_1_word     AT %Q* : WORD; // lampe word to affect to segment color
    Q0001_Balluf_Lampe_1_SycStart AT %Q* : BOOL; // lampe affect to SycStart
    Q0002_Balluf_Lampe_1_SycImp   AT %Q* : BOOL; // lampe affect to SycImp

    //-201A1
    (* Ventil Batterie 201 A*)
    Q0100_14_ST130_kammer_offnen_links     AT %Q* : BOOL; // ST130 Kammer öffnen links
    Q0100_12_                              AT %Q* : BOOL; // 
    Q0101_14_ST130_kammer_offnen_rechts     AT %Q* : BOOL; // ST130 Kammer öffnen rechts
    Q0101_12_                              AT %Q* : BOOL; // 
    Q0102_14_ST130_kammer_nachfullen_links  AT %Q* : BOOL; // ST130 Kammer nachfüllen links
    Q0102_12_                              AT %Q* : BOOL; // 
    Q0103_14_ST130_kammer_nachfullen_rechts AT %Q* : BOOL; // ST130 Kammer nachfüllen rechts
    Q0103_12_                              AT %Q* : BOOL; // 
    Q0104_14_ST130_vibrieren_kammer_links   AT %Q* : BOOL; // ST130 Vibrieren Kammer links/rechts aus
    Q0104_12_ST130_vibrieren_kammer_rechts AT %Q* : BOOL; // ST130 Vibrieren Kammer links/rechts ein
    Q0105_14_ST130_niederhalter_patrone    AT %Q* : BOOL; // ST130 Niederhalter Patrone
    Q0105_12_                              AT %Q* : BOOL; // 
    Q0106_14_ST135_kammer_offnen_links      AT %Q* : BOOL; // ST135 Kammer öffnen links
    Q0106_12_                              AT %Q* : BOOL; // 
    Q0107_14_ST135_kammer_offnen_rechts     AT %Q* : BOOL; // ST135 Kammer öffnen rechts
    Q0107_12_                              AT %Q* : BOOL; // 
    Q0108_14_ST135_kammer_nachfullen_links  AT %Q* : BOOL; // ST135 Kammer nachfüllen links
    Q0108_12_                              AT %Q* : BOOL; // 
    Q0109_14_ST135_kammer_nachfullen_rechts AT %Q* : BOOL; // ST135 Kammer nachfüllen rechts
    Q0109_12_                              AT %Q* : BOOL; // 
    Q0110_14_ST135_vibrieren_kammer_links   AT %Q* : BOOL; // ST135 Vibrieren Kammer links 
    Q0110_12_ST135_vibrieren_kammer_rechts AT %Q* : BOOL; // ST135 Vibrieren Kammer rechts
    Q0111_14_ST135_niederhalter_patrone    AT %Q* : BOOL; // ST135 Niederhalter Patrone
    Q0111_12                               AT %Q* : BOOL; //
    Q0112_14_                               AT %Q* : BOOL; //
    Q0112_12_                              AT %Q* : BOOL; // 
    Q0113_14_                               AT %Q* : BOOL; //
    Q0113_12_                              AT %Q* : BOOL; // 
    Q0114_14_                               AT %Q* : BOOL; //
    Q0114_12_                              AT %Q* : BOOL; // 
    Q0115_14_                               AT %Q* : BOOL; //
    Q0115_12_                              AT %Q* : BOOL; // 

    //-202A1
    (* Ventil Batterie 202 A *)
    Q0200_14_ST145_vakum_greifer_links  AT %Q* : BOOL; // 
    Q0200_12_                           AT %Q* : BOOL; // Vakumgreifer links ST145
    Q0201_14_ST145_vakum_greifer_rechts AT %Q* : BOOL; // 
    Q0201_12_                           AT %Q* : BOOL; // Vakumgreifer rechts ST145
    Q0202_14_ST150_kraftubersetzung     AT %Q* : BOOL; // 
    Q0202_12_                           AT %Q* : BOOL; // Kraftübersetzung ST150
    Q0203_14_ST155_kraftubersetzung     AT %Q* : BOOL; // 
    Q0203_12_                           AT %Q* : BOOL; // Kraftübersetzung ST155
    Q0204_14_                           AT %Q* : BOOL; // 
    Q0204_12_                           AT %Q* : BOOL; // 
    Q0205_14_                           AT %Q* : BOOL; // 
    Q0205_12_                           AT %Q* : BOOL; // 

    //-203A1
    (* Ventil Batterie 203 A *)
    Q0300_14_ST160_niederhalter_links         AT %Q* : BOOL; // ST160 Niederhalter links ST160
    Q0300_12_                                 AT %Q* : BOOL; // 
    Q0301_14_ST160_niederhalter_rechts        AT %Q* : BOOL; // ST160 Niederhalter rechts ST160
    Q0301_12_                                 AT %Q* : BOOL; // 
    Q0302_14_ST160_dichtung_pruflocker_links  AT %Q* : BOOL; // ST160 Dichtung Prüfglocker links
    Q0302_12_ST160_dichtung_pruflocker_rechts AT %Q* : BOOL; // ST160 Dichtung Prüfglocker rechts
    Q0303_14_nc                               AT %Q* : BOOL; // ST160 not connected (yet?)
    Q0303_12_nc                               AT %Q* : BOOL; // ST160 not connected (yet?)
    Q0304_14_ST165_niederhalter_links         AT %Q* : BOOL; // ST165 Niederhalter links ST160   
    Q0304_12_                                 AT %Q* : BOOL; //                                  
    Q0305_14_ST165_niederhalter_rechts        AT %Q* : BOOL; // ST165 Niederhalter rechts ST160  
    Q0305_12_                                 AT %Q* : BOOL; // 
    Q0306_14_ST165_dichtung_pruflocker_links  AT %Q* : BOOL; // ST165 Dichtung Prüfglocker links 
    Q0306_12_ST165_dichtung_pruflocker_rechts AT %Q* : BOOL; // ST165 Dichtung Prüfglocker rechts
    Q0307_14_nc                               AT %Q* : BOOL; // ST165 not connected (yet?)       
    Q0307_12_nc                               AT %Q* : BOOL; // ST165 not connected (yet?)       
    Q0308_14_                                 AT %Q* : BOOL; // 
    Q0308_12_                                 AT %Q* : BOOL; // 
    Q0309_14_                                 AT %Q* : BOOL; // 
    Q0309_12_                                 AT %Q* : BOOL; // 
    Q0310_14_                                 AT %Q* : BOOL; // 
    Q0310_12_                                 AT %Q* : BOOL; // 
    Q0311_14_                                 AT %Q* : BOOL; // 
    Q0311_12_                                 AT %Q* : BOOL; // 

    (* IO-Link Boxen 190A4 *)
    (*******************************************************************)
    //-970B2
    (* FullstandKontrolle ST130.55 *)
    I1000_ AT %I* : BOOL; // FullstandKontrolle ST130.55

    //-970B4
    (* FullstandKontrolle ST130.56 *)
    I1100_ AT %I* : BOOL; // FullstandKontrolle ST130.56

    //-970B6
    (* FullstandKontrolle ST135.55 *)
    I1200_ AT %I* : BOOL; // FullstandKontrolle ST135.55

    //-970B7
    (* FullstandKontrolle ST135.56 *)
    I1300_ AT %I* : BOOL; // 

    //-5009
    (* ST130 I - 8x IO *)
    I1400_ST130_nachfullen_offnen_links_zuruck  AT %I* : BOOL; // 0: Kammer öffnen links zurück
    I1401_ST130_nachfullen_offnen_links_vor     AT %I* : BOOL; // 1: Kammer öffnen links vor
    I1402_ST130_nachfullen_offnen_rechts_zuruck AT %I* : BOOL; // 2: Kammer öffnen rechts zurück
    I1403_ST130_nachfullen_offnen_rechts_vor    AT %I* : BOOL; // 3: Kammer öffnen rechts vor
    I1404_ST130_kammer_offnen_links_zuruck      AT %I* : BOOL; // 4: Kummer nachfüllen links zurück
    I1405_ST130_kammer_offnen_links_vor         AT %I* : BOOL; // 5: Kummer nachfüllen links vor
    I1406_ST130_kammer_offnen_rechts_zuruck     AT %I* : BOOL; // 6: Kammer nachfüllen rechts zurück
    I1407_ST130_kammer_offnen_rechts_vor        AT %I* : BOOL; // 7: Kammer nachfüllen rechts vor

    //-5010
    (* ST135 I - 8x IO *)
    I1500_ST135_nachfullen_offnen_links_zuruck AT %I* : BOOL; // 0: Kammer öffnen links zurück
    I1501_ST135_nachfullen_offnen_rechts_vor   AT %I* : BOOL; // 1: Kammer öffnen links vor
    I1502_ST135_nachfullen_offnen_links_zuruck AT %I* : BOOL; // 2: Kammer öffnen rechts zurück
    I1503_ST135_nachfullen_offnen_rechts_vor   AT %I* : BOOL; // 3: Kammer öffnen rechts vor
    I1504_ST135_kammer_offnen_links_zuruck     AT %I* : BOOL; // 4: Kummer nachfüllen links zurück
    I1505_ST135_kammer_offnen_rechts_vor       AT %I* : BOOL; // 5: Kummer nachfüllen links vor
    I1506_ST135_kammer_offnen_links_zuruck     AT %I* : BOOL; // 6: Kammer nachfüllen rechts zurück
    I1507_ST135_kammer_offnen_rechts_vor       AT %I* : BOOL; // 7: Kammer nachfüllen rechts vor

    //-5014
    (* ST145 I - 4x IO *)
    I1600_ST145_vakum_teil_in_greiffer_left  AT %I* : BOOL; // 0: Vakuumkontrolle Teil in Greifer 145.03
    I1601_ST145_vakum_teil_in_greiffer_right AT %I* : BOOL; // 1: Vakuumkontrolle Teil in Greifer 145.04

    (* IO-Link Boxen 190A8 *)
    (*******************************************************************)
    //-5011
    (* Filterhut vorhanden ST130/135 I - 8x IO *)
    I2000_ST128_filterhut_vorhanden AT %I* : BOOL; // 0: ST130 Filterhut vorhanden links
    //
    I2001_ AT %I* : BOOL; // 
    I2002_ AT %I* : BOOL; // 
    I2003_ AT %I* : BOOL; // 
    I2004_ AT %I* : BOOL; // 
    I2005_ AT %I* : BOOL; // 
    I2006_ AT %I* : BOOL; // 
    I2007_ AT %I* : BOOL; // 

    //-5012
    (* Niederhalter Patrone ST130/135 I - 8x IO *)
    I2100_ST130_niederhalter_patrone_oben  AT %I* : BOOL; // 0: ST130 Niederhalter Patrone oben
    I2101_ST130_niederhalter_patrone_unten AT %I* : BOOL; // 1: ST130 Niederhalter Patrone unten
    I2102_ST135_niederhalter_patrone_oben  AT %I* : BOOL; // 2: ST135 Niederhalter Patrone oben
    I2103_ST135_niederhalter_patrone_unten AT %I* : BOOL; // 3: ST135 Niederhalter Patrone unten

    //-5013
    (* Niederhalter & Vorsatzwanne ST130 I - 8x IO *)
    I2200_ST130_niederhalter_vorne  AT %I* : BOOL; // 0: Niederhalter in Arbeitspos. vorne
    I2201_ST130_niederhalter_hinten AT %I* : BOOL; // 1: Niederhalter in Wartungspos. hinten
    I2202_ST130_Vorsatzwanne_vorne  AT %I* : BOOL; // 2: Vorsatzwanne in Arbeitspos. vorne
    I2203_ST130_Vorsatzwanne_hinten AT %I* : BOOL; // 3: Vorsatzwanne in Ruhepos. hinten

    //-5015
    (* ST145/150/155 I - 8x IO *)
    I2300_ST145_teil_in_vereinzelung    AT %I* : BOOL; // 0: AWK Teil in Vereinzelung (RST) ST145
    I2301_ST150_kraftubersetzung_zuruck AT %I* : BOOL; // 1: Kraftübersetzung zurück ST150
    I2302_ST150_kraftubersetzung_vor    AT %I* : BOOL; // 2: Kraftübersetzung vor ST150
    I2303_ST150_deckel_vohanden         AT %I* : BOOL; // 3: Deckel vorhanden ST150
    I2304_ST155_kraftubersetzung_zuruck AT %I* : BOOL; // 4: Kraftübersetzung zurück ST155
    I2305_ST155_kraftubersetzung_vor    AT %I* : BOOL; // 5: Kraftübersetzung vor ST155
    I2306_ST155_deckel_vohanden         AT %I* : BOOL; // 6: Deckel vorhanden ST155

    //-5501
    (* feeder ST145 *)
    Q2400_ST145_freigabe_REO AT %Q* : BOOL; // 0: Freigabe REO
    I2401_ST145_maximum_wf   AT %I* : BOOL; // 1: Maximum WF
    Q2402_ST145_reigabe_wf   AT %Q* : BOOL; // 2: Freigabe WF

    (* IO-Link Boxen 191A2 *)
    (*******************************************************************)
    //-960B2
    (* Wegmessenor ST160.02 *)
    I3000_ST160_Wegmessenor_links AT %I* : UINT;

    //-960B4
    (* Wegmessenor ST160.03 *)
    I3100_ST160_Wegmessenor_rechts AT %I* : UINT;

    //-960B6
    (* Wegmessenor ST165.02 *)
    I3200_ST165_Wegmessenor_links AT %I* : UINT;

    //-960B7
    (* Wegmessenor ST165.03 *)
    I3300_ST165_Wegmessenor_rechts AT %I* : UINT;

    (*******************************************************************)
    (* EINGÄNGE Schrank B *)
    (*******************************************************************)

    (* IO-Link Boxen 1012045.1 *)
    (*******************************************************************)
    //-10194A3
    (* Meldeleuchte 3 Zonen mit Horni BNI0086 *)
    Q5000_Balluf_Lampe_2_word     AT %Q* : WORD; // lampe word to affect to segment color
    Q5001_Balluf_Lampe_2_SycStart AT %Q* : BOOL; // lampe affect to SycStart
    Q5002_Balluf_Lampe_2_SycImp   AT %Q* : BOOL; // lampe affect to SycImp

    //-10201B1
    (* Ventilbat. 201 B *)
    // empty
    //Q5100_ AT %Q* : BOOL; // eldeleuchte 3 Zonen mit Horni BNI0086

    //-10202B1
    (* Ventilbat. 202 B - 16 slots *)
    Q5200_14_ST115_greifer_links AT %Q* : BOOL; // Greifer links ST115           
    Q5200_12_                    AT %Q* : BOOL; //                               
    Q5201_14_ST115_greifer_rechts           AT %Q* : BOOL; // Greifer rechts ST115          
    Q5201_12_                    AT %Q* : BOOL; //                               
    Q5202_14_ST120_greifer_links            AT %Q* : BOOL; // Greifer links ST120           
    Q5202_12_                    AT %Q* : BOOL; //                               
    Q5203_14_ST120_greifer_rechts           AT %Q* : BOOL; // Greifer rechts ST120          
    Q5203_12_                    AT %Q* : BOOL; //                               
    Q5204_14_ST120_schwenken_links          AT %Q* : BOOL; // Schwenken links ST120         
    Q5204_12_                    AT %Q* : BOOL; //                               
    Q5205_14_ST120_schwenken_rechts         AT %Q* : BOOL; // Schwenken rechts ST120        
    Q5205_12_                    AT %Q* : BOOL; //                               
    Q5206_14_ST125_greifer_filterhut_links  AT %Q* : BOOL; // Greifer Filterhut links ST125 
    Q5206_12_                    AT %Q* : BOOL; //                               
    Q5207_14_ST125_greifer_filterhut_rechts AT %Q* : BOOL; // Greifer Filterhut rechts ST125
    Q5207_12_                    AT %Q* : BOOL; //                               
    Q5208_14_ST125_handling_solerohr_links  AT %Q* : BOOL; // Handling Solerohr links ST125 
    Q5208_12_                    AT %Q* : BOOL; //                               
    Q5209_14_ST125_handling_solerohr_rechts AT %Q* : BOOL; // Handling Solerohr rechts ST125
    Q5209_12_                    AT %Q* : BOOL; //                               
    Q5210_14_ST125_greifer_solerohr_links   AT %Q* : BOOL; // Greifer Solerohr links ST125  
    Q5210_12_                    AT %Q* : BOOL; //                               
    Q5211_14_ST125_greifer_solerohr_rechts  AT %Q* : BOOL; // Greifer Solerohr rechts ST125 
    Q5211_12_                    AT %Q* : BOOL; //                               
    Q5212_14_ST120_stop_vertical_axis AT %Q* : BOOL; // 
    Q5212_12_                    AT %Q* : BOOL; // 
    Q5213_14_                               AT %Q* : BOOL; // 
    Q5213_12_                    AT %Q* : BOOL; // 
    Q5214_14_                               AT %Q* : BOOL; // 
    Q5214_12_                    AT %Q* : BOOL; // 
    Q5215_14_                               AT %Q* : BOOL; // 
    Q5215_12_                    AT %Q* : BOOL; // 

    //-10203B1
    (* Ventilbat. 203 B - 5 slots *)
    Q5300_14_ST175_niederhalter AT %Q* : BOOL; // q0: Niederhalter ST175     
    Q5300_12_                   AT %Q* : BOOL; //                            
    Q5301_14_ST175_kabinentur_einlaufseite AT %Q* : BOOL; // q1: Kabinentür Einlaufseite
    Q5301_12_                   AT %Q* : BOOL; //                            
    Q5302_14_ST175_kabinentur_auflaufseite AT %Q* : BOOL; // q2: Kabinentür Auflaufseite
    Q5302_12_                   AT %Q* : BOOL; //                            
    Q5303_14_                              AT %Q* : BOOL; // q3:                        
    Q5303_12_                   AT %Q* : BOOL; //                            
    Q5304_14_                              AT %Q* : BOOL; // q4:                        
    Q5304_12_                   AT %Q* : BOOL; // 

    //-10204B1
    (* Ventilbat. 204 B - 12 slots *)
    Q5400_14_ST180_greifer_patrone_links AT %Q* : BOOL; // Greifer Patrone links ST180     
    Q5400_12_                            AT %Q* : BOOL; //                                 
    Q5401_14_ST180_greifer_patrone_rechts     AT %Q* : BOOL; // Grefier Patrone rechts ST180    
    Q5401_12_                            AT %Q* : BOOL; //                                 
    Q5402_14_ST180_niederhalter_deckel_links  AT %Q* : BOOL; // Niederhalter Deckel links ST180 
    Q5402_12_                            AT %Q* : BOOL; //                                 
    Q5403_14_ST180_Niederhalter_deckel_rechts AT %Q* : BOOL; // Niederhalter Deckel rechts ST180
    Q5403_12_                            AT %Q* : BOOL; //                                 
    Q5404_14_ST185_greifer_patrone_links      AT %Q* : BOOL; // Greifer Patrone links ST185     
    Q5404_12_                            AT %Q* : BOOL; //                                 
    Q5405_14_ST185_greifer_patrone_rechts     AT %Q* : BOOL; // Greifer Patrone rechts ST185    
    Q5405_12_                            AT %Q* : BOOL; //                                 
    Q5406_14_ST185_niederhalter_deckel_links  AT %Q* : BOOL; // Niederhalter Deckel links ST185 
    Q5406_12_                            AT %Q* : BOOL; //                                 
    Q5407_14_ST185_Niederhalter_deckel_rechts AT %Q* : BOOL; // Niederhalter Deckel rechts ST185
    Q5407_12_                            AT %Q* : BOOL; //                                 
    Q5408_14_ST180_Break_axis_02Z AT %Q* : BOOL; //                                 
    Q5408_12_                            AT %Q* : BOOL; //                                 
    Q5409_14_ST185_Break_axis_02Z AT %Q* : BOOL; //                                 
    Q5409_12_                            AT %Q* : BOOL; // 
    Q5410_14_                                 AT %Q* : BOOL; // 
    Q5410_12_                            AT %Q* : BOOL; // 
    Q5411_14_                                 AT %Q* : BOOL; // 
    Q5411_12_                            AT %Q* : BOOL; // 

    //-10950B1
    (* Vakuumsch. Greifer 110.05 *)
    I5500_ST110_vakumkontrolle_links AT %I* : INT; // Vakuumsch. Greifer 110.05

    //-10950B3
    (* Vakuumsch. Greifer 110.06 *)
    I5600_ST110_vakumkontrolle_rechts AT %I* : INT; // Vakuumsch. Greifer 110.05

    (* IO-Link Boxen 10120A5.2 *)
    (*******************************************************************)
    //-5002
    (* Teil in Vereinzelung (RST) ST110/115 - 8x IO *)
    I6000_ST110_teil_in_vereinzelung AT %I* : BOOL; // Teil in Vereinzelung (RST) ST110
    I6001_ST115_teil_in_vereinzelung AT %I* : BOOL; // Teil in Vereinzelung (RST) ST115

    //-5003
    (* Greifer links ST115 - 4x IO *)
    I6100_ST115_greifer_links_offen       AT %I* : BOOL; // 0: Greifer links offen
    I6101_ST115_greifer_links_geschlossen AT %I* : BOOL; // 1: Greifer links geschlossen

    //-5004
    (* Greifer recht ST115 - 4x IO  *)
    I6200_ST115_greifer_rechts_offen       AT %I* : BOOL; // 0: Greifer rechts offen
    I6201_ST115_greifer_rechts_geschlossen AT %I* : BOOL; // 1: Greifer rechts geschlossen

    //-5005
    (* Greifern link & rechts ST120 - 4x IO*)
    I6300_ST120_greifer_links_geschlossen  AT %I* : BOOL; // 0: Greifer links geschlossen
    I6301_ST120_greifer_links_offen        AT %I* : BOOL; // 1: Greifer links offen
    I6302_ST120_greifer_rechts_geschlossen AT %I* : BOOL; // 2: Greifer rechts geschlossen
    I6303_ST120_greifer_rechts_offen       AT %I* : BOOL; // 3: Greifer rechts offen

    //-5006
    (* feeder ST120 - 8x IO *)
    I6400_ST120_schwenken_links_in_vertikal    AT %I* : BOOL; // 0: Schwenken links vertikal
    I6401_ST120_schwenken_links_in_horizontal  AT %I* : BOOL; // 1: Schwenken links horizontal
    I6402_ST120_schwenken_rechts_in_vertikal   AT %I* : BOOL; // 2: Schwenken rechts vertikal
    I6403_ST120_schwenken_rechts_in_horizontal AT %I* : BOOL; // 3: Schwenken rechts horizontal
    I6404_ST120_teil_in_vereizelung_links      AT %I* : BOOL; // 4: Teil in Vereinzelung links
    I6405_ST120_teil_in_vereinzelung_rechts    AT %I* : BOOL; // 5: Teil in Vereinzelung rechts

    //-5007
    (* Pnp Filterhut Greifer ST125 - 4x IO*)
    I6500_ST125_greiffer_filterhut_links_geschlossen  AT %I* : BOOL; // 0: G. Filterhut links geschlossen
    I6501_ST125_greiffer_filterhut_links_offen        AT %I* : BOOL; // 1: G. Filterhut links offen
    I6502_ST125_greiffer_filterhut_rechts_geschlossen AT %I* : BOOL; // 2: G. Filterhut rechts geschlossen
    I6503_ST125_greiffer_filterhut_rechts_offen       AT %I* : BOOL; // 3: G. Filterhut rechts offen

    //-5008
    (* Pnp Solerohr Greiffer ST125 - 8x IO *)
    I6600_ST125_solerhor_handling_links_unten       AT %I* : BOOL; // 0: Solerohr handling links unten
    I6601_ST125_solerhor_handling_links_oben        AT %I* : BOOL; // 1: Solerohr handling links oben
    I6602_ST125_solerhor_handling_rechts_unten      AT %I* : BOOL; // 2: Solerohr handling rechts unten
    I6603_ST125_solerhor_handling_rechts_oben       AT %I* : BOOL; // 3: Solerohr handling rechts oben
    I6604_ST125_greifer_solerohr_links_geschlossen  AT %I* : BOOL; // 4: G.Solerohr links geschlossen
    I6605_ST125_greifer_solerohr_links_offen        AT %I* : BOOL; // 5: G.Solerohr links offen
    I6606_ST125_greifer_solerohr_rechts_geschlossen AT %I* : BOOL; // 6: G.Solerohr rechts geschlossen
    I6607_ST125_greifer_solerohr_rechts_offen       AT %I* : BOOL; // 7: G.Solerohr rechts offen

    (* IO-Link Boxen 10190A8 *)
    (*******************************************************************)
    //-10945.2 / 110.55
    (* Wandler Kraftsensor 110 links *)
    I7000_ST110_kraftsensor_links AT %I* : BOOL;

    //-10945.3 / 110.56
    (* Wandler Kraftsensor 110 rechts *)
    I7100_ST110_kraftsensor_rechts AT %I* : BOOL;

    //-10945.3 / 115.55
    (* Wandler Kraftsensor 115 links *)
    I7200_ST115_kraftsensor_links AT %I* : BOOL;

    //-10945.5 / 115.56
    (* Wandler Kraftsensor 115 rechts *)
    I7300_ST115_kraftsensor_rechts AT %I* : BOOL;

    //-10945.7 / 120.55
    (* Wandler Kraftsensor 120 links *)
    I7400_ST120_kraftsensor_links AT %I* : BOOL;

    //-10945.8 / 120.56
    (* Wandler Kraftsensor 120 rechts *)
    I7500_ST120_kraftsensor_rechts AT %I* : BOOL;

    //-10946.2 / 125.55
    (* Wandler Kraftsensor 125 links *)
    I7600_ST125_kraftsensor_links AT %I* : BOOL;

    //-10946.3 / 125.56
    (* Wandler Kraftsensor 125 rechts *)
    I7700_ST125_kraftsensor_rechts AT %I* : BOOL;

    (* IO-Link Boxen 10191A2 *)
    (*******************************************************************)
    //-15501
    (* feeder ST110 - 8x IO *)
    Q8000_ST110_freigabe_wf              AT %Q* : BOOL; // 0: Freigabe WF ST110
    I8001_ST110_maximum                  AT %I* : BOOL; // 1: Maximum WF ST110
    I8002_ST110_alarm_forderband         AT %I* : BOOL; // 2: Alarm Förderband ST110
    Q8003_ST110_forderband_ein           AT %Q* : BOOL; // q3: Förderband ein ST110
    I8004_ST110_farbsensor_lagekontrolle AT %I* : BOOL; // 4: Farbsensor Lagekontrolle
    Q8005_ST110_blow_piece               AT %Q* : BOOL; // q5: blow top black pieces into the feeder

    //-15502
    (* feeder ST115 - 8x IO *)
    Q8100_ST115_freigabe_wf      AT %Q* : BOOL; // q0: Freigabe WF ST115
    I8101_ST115_maximum          AT %I* : BOOL; // 1: Maximum WF ST115
    I8102_ST115_alarm_forderband AT %I* : BOOL; // 2: Alarm Förderband ST115
    Q8103_ST115_forderband_ein   AT %Q* : BOOL; // q3: Förderband ein ST115

    //-15503
    (* feeder links ST120 - 8x IO *)
    I8200_ST120_alarm_forderband_l             AT %I* : BOOL; //  0: Alarm Förderband ST115
    Q8201_ST120_forderband_ein_l               AT %Q* : BOOL; // q1: Förderband ein
    I8202_ST120_alarm_forderband_r             AT %I* : BOOL; //  2: Alarm Förderband
    Q8203_ST120_forderband_ein_r               AT %Q* : BOOL; // q3: Förderband ein
    I8204_ST120_hublader_links_unten           AT %I* : BOOL; //  4: Hublader links unten
    I8205_ST120_hublader_links_oben            AT %I* : BOOL; //  5: Hublader links oben
    I8206_ST120_hublader_links_niveaukontrolle AT %I* : BOOL; //  6: Hublader links Nivaukontrolle
    Q8207_ST120_hublader_links_valve           AT %Q* : BOOL; // q7: Hublader links 120.12

    //-15504
    (* feeder rechts ST120 - 8x IO *)
    I8300_ST120_hublader_rechts_unten           AT %I* : BOOL; //  0: Hublader rechts unten
    I8301_ST120_hublader_rechts_oben            AT %I* : BOOL; //  1: Hublader rechts oben
    I8302_ST120_hublader_rechts_niveaukontrolle AT %I* : BOOL; //  2: Hublader rechts Nivaukontrolle
    Q8303_ST120_hublader_rechts_valve           AT %Q* : BOOL; // q3: Hublader rechts 120.13
    I8304_ST120_maxi_zufurung_links             AT %I* : BOOL; //  4: Mini-Maxi Kontrolle Zuführung links
    I8305_ST120_maxi_zufurung_rechts            AT %I* : BOOL; //  5: Mini-Maxi Kontrolle Zuführung rechts

    //-15505
    (* feeder ST125 - 8x IO *)
    Q8400_ST125_freigabe_REO AT %Q* : BOOL; // q0: Freigabe REO
    I8401_ST125_maximum_wf   AT %I* : BOOL; //  1: Maximum WF
    Q8402_ST125_freigabe_wf  AT %Q* : BOOL; // q2: Freigabe WF

    //-5001
    (* feeder ST105 and ST101 - 8x I *)
    I8600_ST105_teil_in_vereinzelung     AT %I* : BOOL; // 1: Teil in Vereinzelung (RST)
    I8601_ST105_shuttle_pin_config_pro   AT %I* : BOOL; // 2: Kontrolle WT-Hülsen Typ Pro
    I8602_ST105_shuttle_pin_config_maxi  AT %I* : BOOL; // 3: Kontrolle WT- Schieber verriegelt
    I8603_ST105_shuttle_ring_pro_present AT %I* : BOOL; // 4: Kontrolle WT- Schieber entriegelt
    I8604_ST105_first_shuttle_pin        AT %I* : BOOL; // 5: Anwesenheit, Init. WT Nr.1

    //-15500
    (* feeder ST105 - 8x IO *)
    I8700_ST105_Ausheber_unten_GS             AT %I* : BOOL; // 1: 
    I8701_ST105_Ausheber_oben_AS              AT %I* : BOOL; // 2: 
    I8702_ST105_Abschieber_zuruck_GS          AT %I* : BOOL; // 3: 
    I8703_ST105_Abschieber_vor_AS             AT %I* : BOOL; // 4: 
    I8704_ST105_Maximum_LF                    AT %I* : BOOL; // 5: 
    I8705_ST105_Kontrolle_zwei_Filtergehiluse AT %I* : BOOL; // 6: 
    I8706_ST105_                              AT %I* : BOOL; // 7: 
    I8707_ST105_                              AT %I* : BOOL; // 8: 

    //-10201B1
    (* Ventilbat. 204 B - 12 slots *)
    Q8800_14_Auschieber_ab_auf     AT %Q* : BOOL; //
	Q8800_12_ AT %Q* : BOOL; // 
    Q8801_14_Auschieber_vor_zuruck AT %Q* : BOOL; // 
	Q8801_12_ AT %Q* : BOOL; // 
    Q8802_14_                      AT %Q* : BOOL; // 
	Q8802_12_ AT %Q* : BOOL; // 
    Q8803_14_                      AT %Q* : BOOL; // 
	Q8803_12_ AT %Q* : BOOL; // 
    Q8804_14_                      AT %Q* : BOOL; // 
	Q8804_12_ AT %Q* : BOOL; // 
    Q8805_14_                      AT %Q* : BOOL; // 
	Q8805_12_ AT %Q* : BOOL; // 

    (* IO-Link Boxen 10191A5 *)
    (*******************************************************************)
    //-5016
    (* ST175/180 8x IO *)
    I9000_ST175_kabinentur_einlauf_offen      AT %I* : BOOL; // 0: Kabinentür Einlauf offen ST175
    I9001_ST175_kabinentur_auslauf_offen      AT %I* : BOOL; // 1: Kabinentür Auslauf offen ST175
    I9002_ST180_entlad_fullstandskontroll_box AT %I* : BOOL; // 2: Entlade-& Füllstandskontrolle Box ST180

    //-5017
    (* pnp ST180 *)
    I9100_ST180_greifer_patrone_links_zu         AT %I* : BOOL; // 0: ST180 Greifer Patrone links zu
    I9101_ST180_greifer_patrone_links_offen      AT %I* : BOOL; // 1: ST180 Greifer Patrone links offen
    I9102_ST180_greifer_patrone_rechts_zu        AT %I* : BOOL; // 2: ST180 Greifer Patrone rechts zu
    I9103_ST180_greifer_patrone_rechts_offen     AT %I* : BOOL; // 3: ST180 Greifer Patrone rechts offen
    I9104_ST180_niederhalter_deckel_links_oben   AT %I* : BOOL; // 4: ST180 Niederhalter Deckel links oben
    I9105_ST180_niederhalter_deckel_links_unten  AT %I* : BOOL; // 5: ST180 Niederhalter Deckel links unten
    I9106_ST180_niederhalter_deckel_rechts_oben  AT %I* : BOOL; // 6: ST180 Niederhalter Deckel rechts oben
    I9107_ST180_niederhalter_deckel_rechts_unten AT %I* : BOOL; // 7: ST180 Niederhalter Deckel rechts unten

    //-5018
    (* pnp ST185 *)
    I9200_ST185_greifer_patrone_links_zu         AT %I* : BOOL; // 0: ST185 Greifer Patrone links zu
    I9201_ST185_greifer_patrone_links_offen      AT %I* : BOOL; // 1: ST185 Greifer Patrone links offen
    I9202_ST185_greifer_patrone_rechts_zu        AT %I* : BOOL; // 2: ST185 Greifer Patrone rechts zu
    I9203_ST185_greifer_patrone_rechts_offen     AT %I* : BOOL; // 3: ST185 Greifer Patrone rechts offen
    I9204_ST185_niederhalter_deckel_links_oben   AT %I* : BOOL; // 4: ST185 Niederhalter Deckel links oben
    I9205_ST185_niederhalter_deckel_links_unten  AT %I* : BOOL; // 5: ST185 Niederhalter Deckel links unten
    I9206_ST185_niederhalter_deckel_rechts_oben  AT %I* : BOOL; // 6: ST185 Niederhalter Deckel rechts oben
    I9207_ST185_niederhalter_deckel_rechts_unten AT %I* : BOOL; // 7: ST185 Niederhalter Deckel rechts unten

    //-10960B2
    (* Wegmesssenor ST175 *)
    I9300_ST175_wegmesssensor AT %I* : UINT; // 0: Wegmesssenor ST175

    //-15506
    (* feeder ST105 *)
    Q9500_ST105_Freigabe_WF         AT %Q* : BOOL; // 1: Run vibrator feeder (nearest of the rotary table)
    Q9501_ST105_Freigabe_LF         AT %Q* : BOOL; // 2 Run LF 
    I9502_ST105_Fullstand_kontrolle AT %I* : BOOL; // 3: vibrator full of piece sensor

END_VAR

// ---- POUs/20_AUTO/BuR SuperTrack com/gMoverAxis.TcGVL
{attribute 'qualified_only'}
VAR_GLOBAL
    I_CT_Shuttle_from_BR AT %I* : CT_Shuttle_BR_to_Tc_u; // all the movers
    Q_CT_Shuttle_to_BR   AT %Q* : CT_Shuttle_Tc_to_BR_u;
    I_CT_Track_from_BR   AT %I* : CT_Track_BR_to_Tc_u;
    Q_CT_Track_to_BR     AT %Q* : CT_Track_Tc_to_BR_u;

END_VAR

// ---- POUs/20_AUTO/ST110/ST110_Axis.TcGVL
{attribute 'qualified_only'}
VAR_GLOBAL CONSTANT
    const110_01Y : AxisLinMotConst_t := (POS_MIN := 0, POS_MAX := 220, VELO_MAX := 1000, VELO_MANU := 100);
    const110_02Z : AxisLinMotConst_t := (POS_MIN := 0, POS_MAX := 200, VELO_MAX := 1500, VELO_MANU := 50);
    const110_03Z : AxisLinMotConst_t := (POS_MIN := 0, POS_MAX := 200, VELO_MAX := 1500, VELO_MANU := 50);
    const110_04Z : AxisLinMotConst_t := (POS_MIN := 0, POS_MAX := 200, VELO_MAX := 1500, VELO_MANU := 50);
    const110_10W : AxisLinMotConst_t := (POS_MIN := 0, POS_MAX := 360, VELO_MAX := 720, VELO_MANU := 50);

END_VAR
VAR_GLOBAL
    axis110_01Y : AxisLinMot_t;
    axis110_02Z : AxisBeckhoff_t;
    axis110_03Z : AxisBeckhoff_t;
    axis110_04Z : AxisBeckhoff_t;
    axis110_10W : AxisLinMot_t;
END_VAR
VAR_GLOBAL RETAIN
    // Recipe values are managed elsewhere
END_VAR

// ---- POUs/20_AUTO/ST115/ST115_Axis.TcGVL
{attribute 'qualified_only'}
VAR_GLOBAL CONSTANT
    const115_01Y : AxisLinMotConst_t := (POS_MIN := -5, POS_MAX := 650, VELO_MAX := 2000, VELO_MANU := 100);
    const115_02Z : AxisLinMotConst_t := (POS_MIN := -5, POS_MAX := 650, VELO_MAX := 2000, VELO_MANU := 50);
    const115_03Z : AxisLinMotConst_t := (POS_MIN := -5, POS_MAX := 650, VELO_MAX := 2000, VELO_MANU := 50);
    const115_04Z : AxisLinMotConst_t := (POS_MIN := -5, POS_MAX := 650, VELO_MAX := 2000, VELO_MANU := 50);
    const115_10W : AxisLinMotConst_t := (POS_MIN := 0, POS_MAX := 360, VELO_MAX := 360, VELO_MANU := 50);

END_VAR
VAR_GLOBAL
    axis115_01Y : AxisLinMot_t;
    axis115_02Z : AxisBeckhoff_t;
    axis115_03Z : AxisBeckhoff_t;
    axis115_04Z : AxisBeckhoff_t;
    axis115_10W : AxisLinMot_t;
END_VAR
VAR_GLOBAL RETAIN
    // Recipe values are managed elsewhere
END_VAR

// ---- POUs/20_AUTO/ST130/ST130_Axis.TcGVL
{attribute 'qualified_only'}
VAR_GLOBAL CONSTANT
    const130_01Z : AxisLinMotConst_t := (POS_MIN := -5, POS_MAX := 245, VELO_MAX := 2000, VELO_MANU := 50);
    const130_10Z : AxisLinMotConst_t := (POS_MIN := -5, POS_MAX := 150, VELO_MAX := 2000, VELO_MANU := 50);

END_VAR
VAR_GLOBAL
    axis130_01Z : AxisBeckhoff_t;
    axis130_10Z : AxisLinMot_t;
END_VAR
VAR_GLOBAL RETAIN
    // Recipe values are managed elsewhere
END_VAR

// ---- POUs/20_AUTO/ST145/ST145_Axis.TcGVL
{attribute 'qualified_only'}
VAR_GLOBAL CONSTANT
    const145_01Y : AxisLinMotConst_t := (POS_MIN := -5, POS_MAX := 200, VELO_MAX := 2000, VELO_MANU := 50);
    const145_02Z : AxisLinMotConst_t := (POS_MIN := -5, POS_MAX := 150, VELO_MAX := 2000, VELO_MANU := 50);
    const145_10W : AxisLinMotConst_t := (POS_MIN := 0, POS_MAX := 360, VELO_MAX := 720, VELO_MANU := 50);

END_VAR
VAR_GLOBAL
    axis145_01Y : AxisLinMot_t;
    axis145_02Z : AxisLinMot_t;
    axis145_10W : AxisLinMot_t;
END_VAR
VAR_GLOBAL RETAIN
    // Recipe values are managed elsewhere
END_VAR

// ---- POUs/20_AUTO/ST170/ST170_Axis.TcGVL
{attribute 'qualified_only'}
VAR_GLOBAL CONSTANT
    const170_01Z : AxisLinMotConst_t := (POS_MIN := 0, POS_MAX := 150, VELO_MAX := 1500, VELO_MANU := 50);

END_VAR
VAR_GLOBAL
    axis170_01Z : AxisLinMot_t;
END_VAR
VAR_GLOBAL RETAIN
    // Recipe values are managed elsewhere
END_VAR

// ---- POUs/20_AUTO/Mover/IProcessSampleMover.TcIO
INTERFACE IProcessSampleMover

METHOD GiveMover : IProcessSampleMover
VAR_INPUT
	mover : REFERENCE TO FB_Mover;
END_VAR
END_METHOD

(* % of completion of the process *)
PROPERTY iCompletionPC : INT
GET
END_GET
END_PROPERTY

PROPERTY Mover : REFERENCE TO FB_Mover
GET
END_GET
SET
END_SET
END_PROPERTY

PROPERTY ProcessExecution : ProcessExecution_e
GET
END_GET
SET
END_SET
END_PROPERTY

METHOD TakeMover : IProcessSampleMover
VAR_INPUT
END_VAR
END_METHOD

METHOD ToString : STRING
VAR_INPUT
END_VAR
END_METHOD

PROPERTY xBusy : BOOL
GET
END_GET
SET
END_SET
END_PROPERTY

PROPERTY xDone : BOOL
GET
END_GET
END_PROPERTY

PROPERTY xMoverPathFree : BOOL
GET
END_GET
END_PROPERTY

PROPERTY xMoverShouldLeave : BOOL
GET
END_GET
END_PROPERTY

END_INTERFACE

// ---- POUs/00_MAIN/MAIN.TcPOU
PROGRAM MAIN
VAR
	MoverMan	: FB_MoverMan;
END_VAR

_02_SAFETY();
_05_FLAGS( xIN_AIR:=TRUE, xIN_btRES_TEMP:=HMI.btArMain[8]);

//HMI
_10_HMI();

MoverMan();

//AUTO
_20_AUTO(xIN_Quit:= _14_STATE._FB_btQUIT.pbtIN^.rtrig , enIN_State:= HMI.enState);

//DJ Test
DEBUG();

END_PROGRAM

// ---- POUs/00_MAIN/_02_SAFETY.TcPOU
PROGRAM _02_SAFETY
(****************************************************************************)
//SAVETY PROGRAMM
//	04.09.2019/Dj
//
//	Version:
(****************************************************************************)
VAR
    //Module
    uiArIN_State AT %I* : ARRAY[1..7] OF UINT; //Module State 
    (* 	1=140D1 
																		2=140D3 
																		3=140D5
																		4=140D7
																		5=140D9
																		6=141D1
																		6=141D3
																		*)
    uiArOUT_State AT %I* : ARRAY[1..3] OF UINT; //Module State 
    (* 	1=141D1 
																		2=141D3 
																		3=141D5
																	*)

    //GR001 IN
    xIN_Reset_bp AT %I* : BOOL;                // blue reset button
    xArIN_Input1 AT %I* : ARRAY[0..7] OF BOOL; //Mapping Inputs 
    xArIN_Input2 AT %I* : ARRAY[0..7] OF BOOL; //Mapping Inputs 
    xArIN_Input3 AT %I* : ARRAY[0..7] OF BOOL; //Mapping Inputs 
    xArIN_Input4 AT %I* : ARRAY[0..7] OF BOOL; //Mapping Inputs 
    xArIN_Input5 AT %I* : ARRAY[0..7] OF BOOL; //Mapping Inputs 
    xArIN_Input6 AT %I* : ARRAY[0..7] OF BOOL; //Mapping Inputs 
    xArIN_Input7 AT %I* : ARRAY[0..7] OF BOOL; //Mapping Inputs 
    (* 	1=140D1 
																		2=140D3 
																		3=140D5
																		4=140D7
																		5=140D9
																		6=141D1
																		7=141D3
																	*)
    //GR002 EStop						
    xIN_ESdelOut AT %I* : BOOL; //EStop del Out
    xIN_ESout    AT %I* : BOOL; //EStop	Out
    xOUT_ResetES AT %Q* : BOOL; //Reset ES

    //GR003 Türen
    xIN_MonDelOut AT %I* : BOOL; //Mon del Out Türen
    xIN_MonOut    AT %I* : BOOL; //Mon Out Türen

    //GR004 AXIS

    //GR005 OUT

    //FB's
    _FB_Gr001Input   : FB_Safety;
    _FB_Gr002NotHalt : FB_Safety;
    _FB_Gr003Tuer    : FB_Safety;
    _FB_Gr004Axis    : FB_Safety;
    _FB_Gr005Output  : FB_Safety;
    _FB_Gr010InputB  : FB_Safety;

END_VAR
VAR_OUTPUT
    xOUT_MonDelOut : BOOL; //Mon del Out
    xOUT_MonOut    : BOOL; //Mon Out	

    xOUT_ESdelOut : BOOL; //EStop del Out
    xOUT_ESout    : BOOL; //EStop Out	

    xOUT_SafetyError     : BOOL; //Error Safety
    xOUT_NotAusBetaetigt : BOOL; //Kein Not-Aus gedrückt
    xOUT_Einrichten      : BOOL; //Einrichten -1-

    XOUT_ST1 : BOOL; //Türe1
    XOUT_ST2 : BOOL; //Türe2
    XOUT_HTA : BOOL; //HubtürA
    XOUT_HTB : BOOL; //HubtürB
    XOUT_HTC : BOOL; //HubtürC
    XOUT_HTD : BOOL; //HubtürD

    XOUT_ESA : BOOL; //NOT-AUS A
    XOUT_ESB : BOOL; //NOT-AUS B
    XOUT_ESC : BOOL; //NOT-AUS C
    XOUT_ESD : BOOL; //NOT-AUS D
    XOUT_ESH : BOOL; //NOT-AUS H
    XOUT_ESP : BOOL; //NOT-AUS Panel
	
	T_RESET : TON;
END_VAR

//--------------------------------------------------------------------------
//SAFETY BAUSTEINE AUFRUFEN
//--------------------------------------------------------------------------	
_FB_Gr001Input(tIN_ResetTime := T#500MS);
_FB_Gr002NotHalt(tIN_ResetTime := T#500MS);
_FB_Gr003Tuer(tIN_ResetTime := T#500MS);
_FB_Gr004Axis(tIN_ResetTime := T#500MS);
_FB_Gr005Output(tIN_ResetTime := T#500MS);
_FB_Gr010InputB(tIN_ResetTime := T#500MS);

//BAUSTEIN ERROR
xOUT_SafetyError := _FB_Gr001Input.xIN_ComErr OR //Gruppe Input
                    _FB_Gr001Input.xIN_FBErr OR
                    _FB_Gr001Input.xIN_OtherErr OR
                    _FB_Gr002NotHalt.xIN_ComErr OR //Gruppe Not-Halt
                    _FB_Gr002NotHalt.xIN_FBErr OR
                    _FB_Gr002NotHalt.xIN_OtherErr OR
                    _FB_Gr003Tuer.xIN_ComErr OR //Gruppe Tür
                    _FB_Gr003Tuer.xIN_FBErr OR
                    _FB_Gr003Tuer.xIN_OtherErr OR
                    _FB_Gr004Axis.xIN_ComErr OR //Gruppe Achsen
                    _FB_Gr004Axis.xIN_FBErr OR
                    _FB_Gr004Axis.xIN_OtherErr OR
                    _FB_Gr005Output.xIN_ComErr OR //Gruppe Output
                    _FB_Gr005Output.xIN_FBErr OR
                    _FB_Gr005Output.xIN_OtherErr OR
                    _FB_Gr001Input.xIN_ComErr OR //Gruppe InputB
                    _FB_Gr001Input.xIN_FBErr OR
                    _FB_Gr001Input.xIN_OtherErr;

//--------------------------------------------------------------------------
//NOT-AUS / ENERGIE ZUUSAMMENFASSUNG
//--------------------------------------------------------------------------	
xOUT_ESdelOut := xIN_ESdelOut;
xOUT_ESOut    := xIN_ESOut;

xOUT_MonDelOut := xIN_MonDelOut;
xOUT_MonOut    := xIN_MonOut;

//--------------------------------------------------------------------------
//NOT-AUS - TÜREN für HMI, TASTEN NICHT ENTRIEGELT	
//--------------------------------------------------------------------------	
//XOUT_ST1 := xArIN_Input5[0] AND xArIN_Input5[1]; //Türe1
//XOUT_ST2 := xArIN_Input5[2] AND
//            xArIN_Input5[3] AND
//            xArIN_Input5[4] AND
//            xArIN_Input5[5]; //Türe2

//XOUT_HTA := xArIN_Input6[0] AND xArIN_Input6[1]; //Hubtüre A
//XOUT_HTB := xArIN_Input6[2] AND xArIN_Input6[3]; //Hubtüre B
//XOUT_HTC := xArIN_Input6[4] AND xArIN_Input6[5]; //Hubtüre C
//XOUT_HTD := xArIN_Input6[6] AND xArIN_Input6[7]; //Hubtüre D
//
//XOUT_ESA := xArIN_Input1[0] AND xArIN_Input1[1]; //NOT-AUS A
//XOUT_ESB := xArIN_Input1[2] AND xArIN_Input1[3]; //NOT-AUS A
//XOUT_ESC := xArIN_Input1[4] AND xArIN_Input1[5]; //NOT-AUS A
//XOUT_ESD := xArIN_Input1[6] AND xArIN_Input1[7]; //NOT-AUS A
//XOUT_ESH := xArIN_Input2[6] AND xArIN_Input2[7]; //NOT-AUS A
//XOUT_ESP := xArIN_Input3[2] AND xArIN_Input3[3]; //NOT-AUS A
//
//xOUT_NotAusBetaetigt := XOUT_ESA AND
//                        XOUT_ESB AND
//                        XOUT_ESC AND
//                        XOUT_ESD AND
//                        XOUT_ESH AND
//                        XOUT_ESP;

//--------------------------------------------------------------------------
//RESET + Einrichten	
//--------------------------------------------------------------------------
T_RESET(IN:=HMI.btArMain[7].button,PT:=T#2S);
xOUT_ResetES    := HMI.Tast_BL OR IN.I_CPX9_1_ResetBp OR T_RESET.Q;
xOUT_Einrichten := xArIN_Input3[1];

////--------------------------------------------------------------------------
////Tür Verriegelung	
////--------------------------------------------------------------------------
//// OUT.Q020_T1_VERR  := (HMI.enState > enState.StateSTEP);
//// OUT.Q021_T2L_VERR := OUT.Q020_T1_VERR;
//// OUT.Q022_T2R_VERR := OUT.Q020_T1_VERR;
//
//xOUT_ESout     := TRUE;
//xOUT_ESdelOut  := TRUE;
//xOUT_MonOut    := TRUE;
//xOUT_MonDelOut := TRUE;
//xOUT_Einrichten := FALSE;  // true when doors are open

END_PROGRAM

// ---- POUs/00_MAIN/DEBUG.TcPOU
PROGRAM DEBUG
VAR
END_VAR

;

END_PROGRAM

// ---- POUs/20_AUTO/FileMan/LoadFromMemory.TcPOU
FUNCTION LoadFromMemory : BOOL
VAR_INPUT
    sData : REFERENCE TO STRING(2000);
END_VAR
VAR
    fbJson     : FB_JsonSaxReader;
    //pJsonParse : FB_ReadJSON;
    //pJsonParse : FB_ReadRecipeJson;

    i : int;
END_VAR

// pJsonParse.myArrayInput1 REF= PERS.iStationTimeDef1;
// pJsonParse.myArrayInput2 REF= PERS.iStationTimeDef2;
//fbJson.Parse(sJson := sData, ipHdl := pJsonParse);

END_FUNCTION

// ---- POUs/20_AUTO/FileMan/ReadJsonDom.TcPOU
FUNCTION ReadJsonDom : BOOL
VAR_INPUT
END_VAR
VAR
    fb_json : FB_JsonDomParser;

    json_head              : SJsonValue;
    json_value             : SJsonValue;
    json_iStationTimeDef1  : SJsonValue;
    json_iStationTimeDef2  : SJsonValue;
    json_recipeList        : SJsonValue;
    json_linearAxis        : SJsonValue;
    json_defProfile        : SJsonValue;
    json_movesList         : SJsonValue;
    json_cylinder2Pos      : SJsonValue;
    json_stationOffsets    : SJsonValue;
    json_st110             : SJsonValue;
    json_FeederConfig      : SJsonValue;
    json_st115             : SJsonValue;
    json_st120             : SJsonValue;
    json_FeederConfigLeft  : SJsonValue;
    json_FeederConfigRight : SJsonValue;
    json_st125             : SJsonValue;
    json_st145             : SJsonValue;
    json_st180             : SJsonValue;
    json_i                 : SJsonValue;
    json_ii                : SJsonValue;
    json_iii               : SJsonValue;

    i   : INT;
    ii  : INT;
    iii : INT;

END_VAR
VAR_IN_OUT
    sMessage : STRING(10000);
END_VAR

json_head := fb_json.ParseDocument(sMessage);

IF fb_json.HasMember(json_head, 'iStationTimeDef1') THEN
    json_iStationTimeDef1 := fb_json.FindMember(json_head, 'iStationTimeDef1');

    IF fb_json.IsArray(json_iStationTimeDef1) THEN
        FOR i := 0 TO MIN(TO_INT(fb_json.GetArraySize(json_iStationTimeDef1)) - 1, CONST.STATION_NUMBER - 1) BY 1 DO
            json_i                       := fb_json.GetArrayValueByIdx(json_iStationTimeDef1, TO_UDINT(i));
            PERS.iStationTimeDef1[i + 1] := TO_DINT(fb_json.GetInt(json_i));
        END_FOR
    END_IF
END_IF

IF fb_json.HasMember(json_head, 'iStationTimeDef2') THEN
    json_iStationTimeDef2 := fb_json.FindMember(json_head, 'iStationTimeDef2');

    IF fb_json.IsArray(json_iStationTimeDef2) THEN
        FOR i := 0 TO MIN(TO_INT(fb_json.GetArraySize(json_iStationTimeDef2)) - 1, CONST.STATION_NUMBER - 1) BY 1 DO
            json_i                       := fb_json.GetArrayValueByIdx(json_iStationTimeDef2, TO_UDINT(i));
            PERS.iStationTimeDef2[i + 1] := TO_DINT(fb_json.GetInt(json_i));
        END_FOR
    END_IF
END_IF

IF fb_json.HasMember(json_head, 'recipeList') THEN
    json_recipeList := fb_json.FindMember(json_head, 'recipeList');

    IF fb_json.IsArray(json_recipeList) THEN
        FOR i := 0 TO MIN(TO_INT(fb_json.GetArraySize(json_recipeList)) - 1, CONST.MAX_RECIPE_NUMBER - 0) BY 1 DO
            json_i := fb_json.GetArrayValueByIdx(json_recipeList, TO_UDINT(i));

            IF fb_json.HasMember(json_i, 'linearAxis') THEN
                json_linearAxis := fb_json.FindMember(json_i, 'linearAxis');

                IF fb_json.IsArray(json_linearAxis) THEN
                    FOR ii := 0 TO MIN(TO_INT(fb_json.GetArraySize(json_linearAxis)) - 1, LinearAxis_e._max - 1 - 0) BY
                        1 DO
                        json_ii := fb_json.GetArrayValueByIdx(json_linearAxis, TO_UDINT(ii));

                        IF fb_json.HasMember(json_ii, 'defProfile') THEN
                            json_defProfile := fb_json.FindMember(json_ii, 'defProfile');

                            IF fb_json.HasMember(json_defProfile, 'lrVelocity') THEN
                                json_value := fb_json.FindMember(json_defProfile, 'lrVelocity');
                                PERS.recipeList[i + 0].linearAxis[ii + 0].defProfile.lrVelocity
                                    := TO_REAL(fb_json.GetDouble(json_value));
                            END_IF

                            IF fb_json.HasMember(json_defProfile, 'lrAccel') THEN
                                json_value := fb_json.FindMember(json_defProfile, 'lrAccel');
                                PERS.recipeList[i + 0].linearAxis[ii + 0].defProfile.lrAccel
                                    := TO_REAL(fb_json.GetDouble(json_value));
                            END_IF

                            IF fb_json.HasMember(json_defProfile, 'lrDecel') THEN
                                json_value := fb_json.FindMember(json_defProfile, 'lrDecel');
                                PERS.recipeList[i + 0].linearAxis[ii + 0].defProfile.lrDecel
                                    := TO_REAL(fb_json.GetDouble(json_value));
                            END_IF

                            IF fb_json.HasMember(json_defProfile, 'lrJerk') THEN
                                json_value := fb_json.FindMember(json_defProfile, 'lrJerk');
                                PERS.recipeList[i + 0].linearAxis[ii + 0].defProfile.lrJerk
                                    := TO_REAL(fb_json.GetDouble(json_value));
                            END_IF
                        END_IF

                        IF fb_json.HasMember(json_ii, 'movesList') THEN
                            json_movesList := fb_json.FindMember(json_ii, 'movesList');

                            IF fb_json.IsArray(json_movesList) THEN
                                FOR iii := 0 TO
                                    MIN(TO_INT(fb_json.GetArraySize(json_movesList)) - 1, CONST.MAX_VECTOR_LIST - 0) BY
                                    1 DO
                                    json_iii := fb_json.GetArrayValueByIdx(json_movesList, TO_UDINT(iii));

                                    IF fb_json.HasMember(json_iii, 'lrVelocity') THEN
                                        json_value := fb_json.FindMember(json_iii, 'lrVelocity');
                                        PERS.recipeList[i + 0].linearAxis[ii + 0].movesList[iii + 0].lrVelocity
                                            := TO_REAL(fb_json.GetDouble(json_value));
                                    END_IF

                                    IF fb_json.HasMember(json_iii, 'lrAccel') THEN
                                        json_value := fb_json.FindMember(json_iii, 'lrAccel');
                                        PERS.recipeList[i + 0].linearAxis[ii + 0].movesList[iii + 0].lrAccel
                                            := TO_REAL(fb_json.GetDouble(json_value));
                                    END_IF

                                    IF fb_json.HasMember(json_iii, 'lrDecel') THEN
                                        json_value := fb_json.FindMember(json_iii, 'lrDecel');
                                        PERS.recipeList[i + 0].linearAxis[ii + 0].movesList[iii + 0].lrDecel
                                            := TO_REAL(fb_json.GetDouble(json_value));
                                    END_IF

                                    IF fb_json.HasMember(json_iii, 'lrJerk') THEN
                                        json_value := fb_json.FindMember(json_iii, 'lrJerk');
                                        PERS.recipeList[i + 0].linearAxis[ii + 0].movesList[iii + 0].lrJerk
                                            := TO_REAL(fb_json.GetDouble(json_value));
                                    END_IF

                                    IF fb_json.HasMember(json_iii, 'lrPosition') THEN
                                        json_value := fb_json.FindMember(json_iii, 'lrPosition');
                                        PERS.recipeList[i + 0].linearAxis[ii + 0].movesList[iii + 0].lrPosition
                                            := TO_LREAL(fb_json.GetDouble(json_value));
                                    END_IF

                                    IF fb_json.HasMember(json_iii, 'TriggerType') THEN
                                        json_value := fb_json.FindMember(json_iii, 'TriggerType');
                                        PERS.recipeList[i + 0].linearAxis[ii + 0].movesList[iii + 0].TriggerType
                                            := TO_INT(fb_json.GetInt(json_value));
                                    END_IF

                                    IF fb_json.HasMember(json_iii, 'TriggerPos') THEN
                                        json_value := fb_json.FindMember(json_iii, 'TriggerPos');
                                        PERS.recipeList[i + 0].linearAxis[ii + 0].movesList[iii + 0].TriggerPos
                                            := TO_LREAL(fb_json.GetDouble(json_value));
                                    END_IF

                                    IF fb_json.HasMember(json_iii, 'Timeout_ms') THEN
                                        json_value := fb_json.FindMember(json_iii, 'Timeout_ms');
                                        PERS.recipeList[i + 0].linearAxis[ii + 0].movesList[iii + 0].Timeout_ms
                                            := TO_DINT(fb_json.GetInt(json_value));
                                    END_IF
                                END_FOR
                            END_IF
                        END_IF
                    END_FOR
                END_IF
            END_IF

            IF fb_json.HasMember(json_i, 'cylinder2Pos') THEN
                json_cylinder2Pos := fb_json.FindMember(json_i, 'cylinder2Pos');

                IF fb_json.IsArray(json_cylinder2Pos) THEN
                    FOR ii := 0 TO MIN(TO_INT(fb_json.GetArraySize(json_cylinder2Pos)) - 1, StationList_e._max - 1) BY
                        1 DO
                        json_ii := fb_json.GetArrayValueByIdx(json_cylinder2Pos, TO_UDINT(ii));

                        IF fb_json.IsArray(json_ii) THEN
                            FOR iii := 0 TO
                                MIN(TO_INT(fb_json.GetArraySize(json_ii)) - 1, CONST.MAX_CYLINDER_PER_STATION - 1) BY
                                1 DO
                                json_iii := fb_json.GetArrayValueByIdx(json_ii, TO_UDINT(iii));

                                IF fb_json.HasMember(json_iii, 'toGS_alarm_time') THEN
                                    json_value := fb_json.FindMember(json_iii, 'toGS_alarm_time');
                                    PERS.recipeList[i + 0].cylinder2Pos[ii + 0][iii + 0].toGS_alarm_time
                                        := TO_DINT(fb_json.GetInt(json_value));
                                END_IF

                                IF fb_json.HasMember(json_iii, 'toAS_alarm_time') THEN
                                    json_value := fb_json.FindMember(json_iii, 'toAS_alarm_time');
                                    PERS.recipeList[i + 0].cylinder2Pos[ii + 0][iii + 0].toAS_alarm_time
                                        := TO_DINT(fb_json.GetInt(json_value));
                                END_IF

                                IF fb_json.HasMember(json_iii, 'toGS_wait_time') THEN
                                    json_value := fb_json.FindMember(json_iii, 'toGS_wait_time');
                                    PERS.recipeList[i + 0].cylinder2Pos[ii + 0][iii + 0].toGS_wait_time
                                        := TO_DINT(fb_json.GetInt(json_value));
                                END_IF

                                IF fb_json.HasMember(json_iii, 'toAS_wait_time') THEN
                                    json_value := fb_json.FindMember(json_iii, 'toAS_wait_time');
                                    PERS.recipeList[i + 0].cylinder2Pos[ii + 0][iii + 0].toAS_wait_time
                                        := TO_DINT(fb_json.GetInt(json_value));
                                END_IF
                            END_FOR
                        END_IF
                    END_FOR
                END_IF

                IF fb_json.HasMember(json_i, 'stationOffsets') THEN
                    json_stationOffsets := fb_json.FindMember(json_i, 'stationOffsets');

                    IF fb_json.IsArray(json_stationOffsets) THEN
                        FOR ii := 0 TO
                            MIN(TO_INT(fb_json.GetArraySize(json_stationOffsets)) - 1, CONST.STATION_NUMBER - 1 - 0) BY
                            1 DO
                            json_ii := fb_json.GetArrayValueByIdx(json_stationOffsets, TO_UDINT(ii));
                            PERS.recipeList[i + 0].stationOffsets[ii + 0]
                                := TO_REAL(fb_json.GetDouble(json_ii));
                        END_FOR
                    END_IF
                END_IF

                IF fb_json.HasMember(json_i, 'st110') THEN
                    json_st110 := fb_json.FindMember(json_i, 'st110');

                    IF fb_json.HasMember(json_st110, 'xUseVerLeft') THEN
                        json_value                               := fb_json.FindMember(json_st110, 'xUseVerLeft');
                        PERS.recipeList[i + 0].st110.xUseVerLeft := (fb_json.GetBool(json_value));
                    END_IF

                    IF fb_json.HasMember(json_st110, 'xUseVerRight') THEN
                        json_value                                := fb_json.FindMember(json_st110, 'xUseVerRight');
                        PERS.recipeList[i + 0].st110.xUseVerRight := (fb_json.GetBool(json_value));
                    END_IF

                    IF fb_json.HasMember(json_st110, 'FeederConfig') THEN
                        json_FeederConfig := fb_json.FindMember(json_st110, 'FeederConfig');

                        IF fb_json.HasMember(json_FeederConfig, 'InFilterDelay') THEN
                            json_value := fb_json.FindMember(json_FeederConfig, 'InFilterDelay');
                            PERS.recipeList[i + 0].st110.FeederConfig.InFilterDelay
                                := TO_DINT(fb_json.GetInt(json_value));
                        END_IF

                        IF fb_json.HasMember(json_FeederConfig, 'StartDelay') THEN
                            json_value := fb_json.FindMember(json_FeederConfig, 'StartDelay');
                            PERS.recipeList[i + 0].st110.FeederConfig.StartDelay
                                := TO_DINT(fb_json.GetInt(json_value));
                        END_IF

                        IF fb_json.HasMember(json_FeederConfig, 'StopDelay') THEN
                            json_value := fb_json.FindMember(json_FeederConfig, 'StopDelay');
                            PERS.recipeList[i + 0].st110.FeederConfig.StopDelay
                                := TO_DINT(fb_json.GetInt(json_value));
                        END_IF

                        IF fb_json.HasMember(json_FeederConfig, 'EmptyDelay') THEN
                            json_value := fb_json.FindMember(json_FeederConfig, 'EmptyDelay');
                            PERS.recipeList[i + 0].st110.FeederConfig.EmptyDelay
                                := TO_DINT(fb_json.GetInt(json_value));
                        END_IF
                    END_IF
                END_IF

                IF fb_json.HasMember(json_i, 'st115') THEN
                    json_st115 := fb_json.FindMember(json_i, 'st115');

                    IF fb_json.HasMember(json_st115, 'xUseVerLeft') THEN
                        json_value                               := fb_json.FindMember(json_st115, 'xUseVerLeft');
                        PERS.recipeList[i + 0].st115.xUseVerLeft := (fb_json.GetBool(json_value));
                    END_IF

                    IF fb_json.HasMember(json_st115, 'xUseVerRight') THEN
                        json_value                                := fb_json.FindMember(json_st115, 'xUseVerRight');
                        PERS.recipeList[i + 0].st115.xUseVerRight := (fb_json.GetBool(json_value));
                    END_IF

                    IF fb_json.HasMember(json_st115, 'FeederConfig') THEN
                        json_FeederConfig := fb_json.FindMember(json_st115, 'FeederConfig');

                        IF fb_json.HasMember(json_FeederConfig, 'InFilterDelay') THEN
                            json_value := fb_json.FindMember(json_FeederConfig, 'InFilterDelay');
                            PERS.recipeList[i + 0].st115.FeederConfig.InFilterDelay
                                := TO_DINT(fb_json.GetInt(json_value));
                        END_IF

                        IF fb_json.HasMember(json_FeederConfig, 'StartDelay') THEN
                            json_value := fb_json.FindMember(json_FeederConfig, 'StartDelay');
                            PERS.recipeList[i + 0].st115.FeederConfig.StartDelay
                                := TO_DINT(fb_json.GetInt(json_value));
                        END_IF

                        IF fb_json.HasMember(json_FeederConfig, 'StopDelay') THEN
                            json_value := fb_json.FindMember(json_FeederConfig, 'StopDelay');
                            PERS.recipeList[i + 0].st115.FeederConfig.StopDelay
                                := TO_DINT(fb_json.GetInt(json_value));
                        END_IF

                        IF fb_json.HasMember(json_FeederConfig, 'EmptyDelay') THEN
                            json_value := fb_json.FindMember(json_FeederConfig, 'EmptyDelay');
                            PERS.recipeList[i + 0].st115.FeederConfig.EmptyDelay
                                := TO_DINT(fb_json.GetInt(json_value));
                        END_IF
                    END_IF
                END_IF

                IF fb_json.HasMember(json_i, 'st120') THEN
                    json_st120 := fb_json.FindMember(json_i, 'st120');

                    IF fb_json.HasMember(json_st120, 'xUseVerLeft') THEN
                        json_value                               := fb_json.FindMember(json_st120, 'xUseVerLeft');
                        PERS.recipeList[i + 0].st120.xUseVerLeft := (fb_json.GetBool(json_value));
                    END_IF

                    IF fb_json.HasMember(json_st120, 'xUseVerRight') THEN
                        json_value                                := fb_json.FindMember(json_st120, 'xUseVerRight');
                        PERS.recipeList[i + 0].st120.xUseVerRight := (fb_json.GetBool(json_value));
                    END_IF

                    IF fb_json.HasMember(json_st120, 'FeederConfigLeft') THEN
                        json_FeederConfigLeft := fb_json.FindMember(json_st120, 'FeederConfigLeft');

                        IF fb_json.HasMember(json_FeederConfigLeft, 'InFilterDelay') THEN
                            json_value := fb_json.FindMember(json_FeederConfigLeft, 'InFilterDelay');
                            PERS.recipeList[i + 0].st120.FeederConfigLeft.InFilterDelay
                                := TO_DINT(fb_json.GetInt(json_value));
                        END_IF

                        IF fb_json.HasMember(json_FeederConfigLeft, 'StartDelay') THEN
                            json_value := fb_json.FindMember(json_FeederConfigLeft, 'StartDelay');
                            PERS.recipeList[i + 0].st120.FeederConfigLeft.StartDelay
                                := TO_DINT(fb_json.GetInt(json_value));
                        END_IF

                        IF fb_json.HasMember(json_FeederConfigLeft, 'StopDelay') THEN
                            json_value := fb_json.FindMember(json_FeederConfigLeft, 'StopDelay');
                            PERS.recipeList[i + 0].st120.FeederConfigLeft.StopDelay
                                := TO_DINT(fb_json.GetInt(json_value));
                        END_IF

